KUKA KRL program: EPS_2_251674_SAN01_A_20251204014854.src

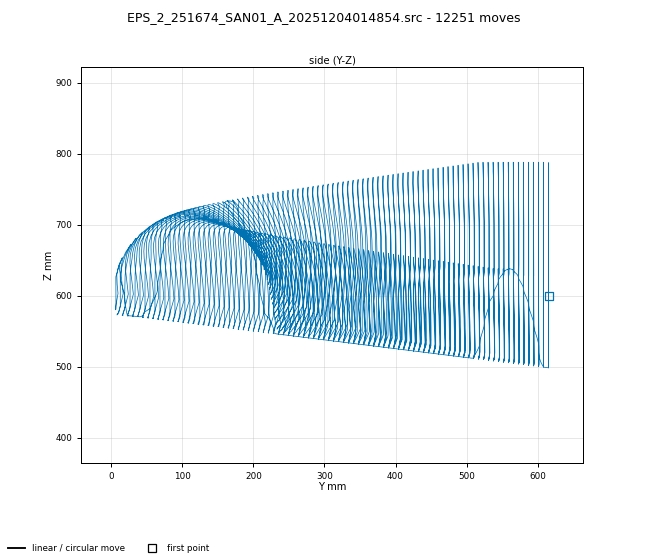
[picture p0: tool path of EPS_2_251674_SAN01_A_20251204014854.src, 12251 of 12253 moves have a stored position in this frame; points joined in program order, loops and branches not executed]
&ACCESS RVP
&REL 4
&COMMENT QRS 19112012
&PARAM EDITMASK = *
DEF PART()
EXT BAS (BAS_COMMAND :IN,REAL :IN )
INT I
BAS (#INITMOV,0 )

;KUKA QRS Post kuka4.cps  Date:22-06-2017 !

File_ID=2937

QRS_PRE_INIT()

;Init var - Until changes are made in qrs_pre_init
Outlet_Square_prg=0
Inlet_1_Square_prg=0
Inlet_2_Square_prg=0
Inlet_3_Square_prg=0
Inlet_4_Square_prg=0
Inlet_5_Square_prg=0

Outlet_1={X 0.000, Y 519.550, Z 713.000, B 0.000, E1 0.000 }
Inlet_1={X 0.000, Y 537.700, Z 427.500, B 0.000, E1 111.000 }
Outlet_1_type=150
Inlet_1_type=201
;QRS#1=Sidecore dimensions
;QRS#2=150-6" PVC SDR 28
;QRS#3=200-8" PVC SDR 35
;QRS#4=
;QRS#5=
;QRS#6=
;QRS#7=
;QRS#8=
;QRS#9=10-06 PSX
;QRS#10=12-08 PSX
;QRS#11=
;QRS#12=
;QRS#13=
;QRS#14=
;QRS#15=
;QRS#16=1220x127x1067 3,5'
;QRS#17=EPS Height
;QRS#18=788
;QRS#19=*
;QRS#20= UPDATED VERSION 22-06-2017
;QRS#21=*
Outlet_Square=070
Inlet_1_Square=0100
Inlet_2_Square=0
Inlet_3_Square=0
Inlet_4_Square=0
Inlet_5_Square=0
Mill_Square=1
Outlet_Square_Prg=203
Inlet_1_Square_prg=204

QRS_INIT()

$ADVANCE=5

; T1
PTP {E1 173.59,E2 173.59}
PTP {X 0,Y 615.512,A -85,B 0,C 180,E1 173.59,E2 173.59,E3 0,E4 0,E5 0,E6 0}
QRS_SPEED_INIT()
LIN {X 0,Y 615.512,Z 600,A -85,B 0,C 180,E1 173.59,E2 173.59,E3 0,E4 0,E5 0,E6 0} C_VEL
LIN {X 0,Y 615.512,Z 508.679,A -85,B 0,C 180,E1 173.59,E2 173.59} C_VEL
LIN {X 0,Y 615.512,Z 500.505,A -85,B 0,C 180,E1 173.59,E2 173.59} C_VEL
LIN {X 0,Y 615.495,Z 498.505,A -85,B 0,C 180,E1 173.404,E2 173.404} C_VEL
LIN {X 0,Y 615.498,Z 498.684,A -85,B 0,C 180,E1 171.091,E2 171.091} C_VEL
LIN {X 0,Y 615.497,Z 499.843,A -85,B 0,C 180,E1 170.967,E2 170.967} C_VEL
LIN {X 0,Y 615.499,Z 535.633,A -85,B 0,C 180,E1 170.511,E2 170.511} C_VEL
LIN {X 0,Y 615.498,Z 548.242,A -85,B 0,C 180,E1 170.221,E2 170.221} C_VEL
LIN {X 0,Y 615.498,Z 560.585,A -85,B 0,C 180,E1 169.806,E2 169.806} C_VEL
LIN {X 0,Y 615.498,Z 572.014,A -85,B 0,C 180,E1 169.287,E2 169.287} C_VEL
LIN {X 0,Y 615.494,Z 583.164,A -85,B 0,C 180,E1 168.64,E2 168.64} C_VEL
LIN {X 0,Y 615.498,Z 593.556,A -85,B 0,C 180,E1 167.888,E2 167.888} C_VEL
LIN {X 0,Y 615.498,Z 602.092,A -85,B 0,C 180,E1 167.134,E2 167.134} C_VEL
LIN {X 0,Y 615.498,Z 611.332,A -85,B 0,C 180,E1 166.126,E2 166.126} C_VEL
LIN {X 0,Y 615.498,Z 618.787,A -85,B 0,C 180,E1 165.113,E2 165.113} C_VEL
LIN {X 0,Y 615.496,Z 624.756,A -85,B 0,C 180,E1 164.095,E2 164.095} C_VEL
LIN {X 0,Y 615.496,Z 629.436,A -85,B 0,C 180,E1 163.072,E2 163.072} C_VEL
LIN {X 0,Y 615.495,Z 632.975,A -85,B 0,C 180,E1 162.043,E2 162.043} C_VEL
LIN {X 0,Y 615.497,Z 634.719,A -85,B 0,C 180,E1 161.354,E2 161.354} C_VEL
LIN {X 0,Y 615.495,Z 636.035,A -85,B 0,C 180,E1 160.662,E2 160.662} C_VEL
LIN {X 0,Y 615.493,Z 637.28,A -85,B 0,C 180,E1 159.438,E2 159.438} C_VEL
LIN {X 0,Y 615.499,Z 637.302,A -85,B 0,C 180,E1 158.568,E2 158.568} C_VEL
LIN {X 0,Y 615.491,Z 636.585,A -85,B 0,C 180,E1 157.65,E2 157.65} C_VEL
LIN {X 0,Y 615.494,Z 634.477,A -85,B 0,C 180,E1 156.444,E2 156.444} C_VEL
LIN {X 0,Y 615.496,Z 631.396,A -85,B 0,C 180,E1 155.369,E2 155.369} C_VEL
LIN {X 0,Y 615.494,Z 627.053,A -85,B 0,C 180,E1 154.284,E2 154.284} C_VEL
LIN {X 0,Y 615.498,Z 621.628,A -85,B 0,C 180,E1 153.254,E2 153.254} C_VEL
LIN {X 0,Y 615.494,Z 615.11,A -85,B 0,C 180,E1 152.27,E2 152.27} C_VEL
LIN {X 0,Y 615.497,Z 607.528,A -85,B 0,C 180,E1 151.342,E2 151.342} C_VEL
LIN {X 0,Y 615.498,Z 599.104,A -85,B 0,C 180,E1 150.496,E2 150.496} C_VEL
LIN {X 0,Y 615.495,Z 588.703,A -85,B 0,C 180,E1 149.651,E2 149.651} C_VEL
LIN {X 0,Y 615.497,Z 577.291,A -85,B 0,C 180,E1 148.91,E2 148.91} C_VEL
LIN {X 0,Y 615.498,Z 565.584,A -85,B 0,C 180,E1 148.315,E2 148.315} C_VEL
LIN {X 0,Y 615.496,Z 552.815,A -85,B 0,C 180,E1 147.828,E2 147.828} C_VEL
LIN {X 0,Y 615.497,Z 539.404,A -85,B 0,C 180,E1 147.47,E2 147.47} C_VEL
LIN {X 0,Y 615.497,Z 525.299,A -85,B 0,C 180,E1 147.251,E2 147.251} C_VEL
LIN {X 0,Y 615.496,Z 499.662,A -85,B 0,C 180,E1 146.935,E2 146.935} C_VEL
LIN {X 0,Y 615.495,Z 498.663,A -85,B 0,C 180,E1 146.813,E2 146.813} C_VEL
LIN {X 0,Y 615.487,Z 498.499,A -85,B 0,C 180,E1 144.164,E2 144.164} C_VEL
LIN {X 0,Y 615.478,Z 498.497,A -85,B 0,C 180,E1 141.93,E2 141.93} C_VEL
LIN {X 0,Y 615.482,Z 498.497,A -85,B 0,C 180,E1 139.393,E2 139.393} C_VEL
LIN {X 0,Y 615.485,Z 498.512,A -85,B 0,C 180,E1 136.755,E2 136.755} C_VEL
LIN {X 0,Y 615.482,Z 498.498,A -85,B 0,C 180,E1 133.996,E2 133.996} C_VEL
LIN {X 0,Y 615.483,Z 498.495,A -85,B 0,C 180,E1 131.473,E2 131.473} C_VEL
LIN {X 0,Y 615.482,Z 498.505,A -85,B 0,C 180,E1 128.904,E2 128.904} C_VEL
LIN {X 0,Y 615.491,Z 498.509,A -85,B 0,C 180,E1 126.423,E2 126.423} C_VEL
LIN {X 0,Y 615.479,Z 498.496,A -85,B 0,C 180,E1 123.532,E2 123.532} C_VEL
LIN {X 0,Y 615.48,Z 498.503,A -85,B 0,C 180,E1 120.919,E2 120.919} C_VEL
LIN {X 0,Y 615.496,Z 498.512,A -85,B 0,C 180,E1 118.451,E2 118.451} C_VEL
LIN {X 0,Y 615.477,Z 498.496,A -85,B 0,C 180,E1 115.566,E2 115.566} C_VEL
LIN {X 0,Y 615.482,Z 498.503,A -85,B 0,C 180,E1 112.844,E2 112.844} C_VEL
LIN {X 0,Y 615.489,Z 498.502,A -85,B 0,C 180,E1 110.032,E2 110.032} C_VEL
LIN {X 0,Y 615.485,Z 498.495,A -85,B 0,C 180,E1 107.27,E2 107.27} C_VEL
LIN {X 0,Y 615.484,Z 498.51,A -85,B 0,C 180,E1 104.549,E2 104.549} C_VEL
LIN {X 0,Y 615.485,Z 498.5,A -85,B 0,C 180,E1 101.861,E2 101.861} C_VEL
LIN {X 0,Y 615.486,Z 498.495,A -85,B 0,C 180,E1 99.199,E2 99.199} C_VEL
LIN {X 0,Y 615.477,Z 498.509,A -85,B 0,C 180,E1 96.557,E2 96.557} C_VEL
LIN {X 0,Y 615.487,Z 498.503,A -85,B 0,C 180,E1 93.928,E2 93.928} C_VEL
LIN {X 0,Y 615.48,Z 498.496,A -85,B 0,C 180,E1 91.309,E2 91.309} C_VEL
LIN {X 0,Y 615.483,Z 498.502,A -85,B 0,C 180,E1 88.691,E2 88.691} C_VEL
LIN {X 0,Y 615.496,Z 498.507,A -85,B 0,C 180,E1 86.072,E2 86.072} C_VEL
LIN {X 0,Y 615.477,Z 498.497,A -85,B 0,C 180,E1 83.435,E2 83.435} C_VEL
LIN {X 0,Y 615.486,Z 498.497,A -85,B 0,C 180,E1 80.801,E2 80.801} C_VEL
LIN {X 0,Y 615.489,Z 498.514,A -85,B 0,C 180,E1 78.139,E2 78.139} C_VEL
LIN {X 0,Y 615.476,Z 498.499,A -85,B 0,C 180,E1 75.451,E2 75.451} C_VEL
LIN {X 0,Y 615.485,Z 498.498,A -85,B 0,C 180,E1 72.73,E2 72.73} C_VEL
LIN {X 0,Y 615.495,Z 498.509,A -85,B 0,C 180,E1 69.968,E2 69.968} C_VEL
LIN {X 0,Y 615.48,Z 498.496,A -85,B 0,C 180,E1 67.156,E2 67.156} C_VEL
LIN {X 0,Y 615.479,Z 498.504,A -85,B 0,C 180,E1 64.434,E2 64.434} C_VEL
LIN {X 0,Y 615.487,Z 498.513,A -85,B 0,C 180,E1 62.086,E2 62.086} C_VEL
LIN {X 0,Y 615.499,Z 498.506,A -85,B 0,C 180,E1 59.841,E2 59.841} C_VEL
LIN {X 0,Y 615.481,Z 498.502,A -85,B 0,C 180,E1 57.543,E2 57.543} C_VEL
LIN {X 0,Y 615.478,Z 498.497,A -85,B 0,C 180,E1 55.185,E2 55.185} C_VEL
LIN {X 0,Y 615.491,Z 498.494,A -85,B 0,C 180,E1 52.759,E2 52.759} C_VEL
LIN {X 0,Y 615.497,Z 498.513,A -85,B 0,C 180,E1 49.911,E2 49.911} C_VEL
LIN {X 0,Y 615.485,Z 498.494,A -85,B 0,C 180,E1 46.953,E2 46.953} C_VEL
LIN {X 0,Y 615.478,Z 498.508,A -85,B 0,C 180,E1 44.151,E2 44.151} C_VEL
LIN {X 0,Y 615.482,Z 498.503,A -85,B 0,C 180,E1 41.475,E2 41.475} C_VEL
LIN {X 0,Y 615.484,Z 498.495,A -85,B 0,C 180,E1 38.905,E2 38.905} C_VEL
LIN {X 0,Y 615.481,Z 498.499,A -85,B 0,C 180,E1 36.426,E2 36.426} C_VEL
LIN {X 0,Y 615.486,Z 498.506,A -85,B 0,C 180,E1 33.536,E2 33.536} C_VEL
LIN {X 0,Y 615.483,Z 498.495,A -85,B 0,C 180,E1 30.92,E2 30.92} C_VEL
LIN {X 0,Y 615.483,Z 498.497,A -85,B 0,C 180,E1 28.452,E2 28.452} C_VEL
LIN {X 0,Y 615.493,Z 498.508,A -85,B 0,C 180,E1 25.573,E2 25.573} C_VEL
LIN {X 0,Y 615.482,Z 498.496,A -85,B 0,C 180,E1 22.845,E2 22.845} C_VEL
LIN {X 0,Y 615.477,Z 498.505,A -85,B 0,C 180,E1 20.033,E2 20.033} C_VEL
LIN {X 0,Y 615.479,Z 498.504,A -85,B 0,C 180,E1 17.271,E2 17.271} C_VEL
LIN {X 0,Y 615.488,Z 498.494,A -85,B 0,C 180,E1 14.549,E2 14.549} C_VEL
LIN {X 0,Y 615.479,Z 498.508,A -85,B 0,C 180,E1 11.861,E2 11.861} C_VEL
LIN {X 0,Y 615.479,Z 498.504,A -85,B 0,C 180,E1 9.199,E2 9.199} C_VEL
LIN {X 0,Y 615.491,Z 498.493,A -85,B 0,C 180,E1 6.557,E2 6.557} C_VEL
LIN {X 0,Y 615.475,Z 498.505,A -85,B 0,C 180,E1 3.929,E2 3.929} C_VEL
LIN {X 0,Y 615.484,Z 498.508,A -85,B 0,C 180,E1 1.309,E2 1.309} C_VEL
LIN {X 0,Y 615.485,Z 498.495,A -85,B 0,C 180,E1 -1.308,E2 -1.308} C_VEL
LIN {X 0,Y 615.477,Z 498.5,A -85,B 0,C 180,E1 -3.928,E2 -3.928} C_VEL
LIN {X 0,Y 615.49,Z 498.513,A -85,B 0,C 180,E1 -6.591,E2 -6.591} C_VEL
LIN {X 0,Y 615.479,Z 498.499,A -85,B 0,C 180,E1 -9.199,E2 -9.199} C_VEL
LIN {X 0,Y 615.479,Z 498.497,A -85,B 0,C 180,E1 -11.861,E2 -11.861} C_VEL
LIN {X 0,Y 615.488,Z 498.513,A -85,B 0,C 180,E1 -14.549,E2 -14.549} C_VEL
LIN {X 0,Y 615.478,Z 498.499,A -85,B 0,C 180,E1 -17.271,E2 -17.271} C_VEL
LIN {X 0,Y 615.477,Z 498.499,A -85,B 0,C 180,E1 -20.033,E2 -20.033} C_VEL
LIN {X 0,Y 615.482,Z 498.51,A -85,B 0,C 180,E1 -22.845,E2 -22.845} C_VEL
LIN {X 0,Y 615.493,Z 498.493,A -85,B 0,C 180,E1 -25.715,E2 -25.715} C_VEL
LIN {X 0,Y 615.487,Z 498.513,A -85,B 0,C 180,E1 -28.658,E2 -28.658} C_VEL
LIN {X 0,Y 615.478,Z 498.505,A -85,B 0,C 180,E1 -31.087,E2 -31.087} C_VEL
LIN {X 0,Y 615.485,Z 498.496,A -85,B 0,C 180,E1 -33.536,E2 -33.536} C_VEL
LIN {X 0,Y 615.486,Z 498.494,A -85,B 0,C 180,E1 -35.835,E2 -35.835} C_VEL
LIN {X 0,Y 615.478,Z 498.498,A -85,B 0,C 180,E1 -38.069,E2 -38.069} C_VEL
LIN {X 0,Y 615.482,Z 498.508,A -85,B 0,C 180,E1 -40.607,E2 -40.607} C_VEL
LIN {X 0,Y 615.477,Z 498.504,A -85,B 0,C 180,E1 -43.245,E2 -43.245} C_VEL
LIN {X 0,Y 615.482,Z 498.495,A -85,B 0,C 180,E1 -46.003,E2 -46.003} C_VEL
LIN {X 0,Y 615.483,Z 498.504,A -85,B 0,C 180,E1 -48.527,E2 -48.527} C_VEL
LIN {X 0,Y 615.479,Z 498.51,A -85,B 0,C 180,E1 -51.096,E2 -51.096} C_VEL
LIN {X 0,Y 615.484,Z 498.497,A -85,B 0,C 180,E1 -53.576,E2 -53.576} C_VEL
LIN {X 0,Y 615.479,Z 498.502,A -85,B 0,C 180,E1 -56.467,E2 -56.467} C_VEL
LIN {X 0,Y 615.477,Z 498.514,A -85,B 0,C 180,E1 -59.08,E2 -59.08} C_VEL
LIN {X 0,Y 615.482,Z 498.5,A -85,B 0,C 180,E1 -61.551,E2 -61.551} C_VEL
LIN {X 0,Y 615.495,Z 498.704,A -85,B 0,C 180,E1 -63.104,E2 -63.104} C_VEL
LIN {X 0,Y 615.495,Z 501.655,A -85,B 0,C 180,E1 -63.557,E2 -63.557} C_VEL
LIN {X 0,Y 615.481,Z 521.157,A -85,B 0,C 180,E1 -66.217,E2 -66.217} C_VEL
LIN {X 0,Y 615.497,Z 541.369,A -85,B 0,C 180,E1 -68.92,E2 -68.92} C_VEL
LIN {X 0,Y 615.492,Z 563.931,A -85,B 0,C 180,E1 -71.882,E2 -71.882} C_VEL
LIN {X 0,Y 615.489,Z 586.305,A -85,B 0,C 180,E1 -74.774,E2 -74.774} C_VEL
LIN {X 0,Y 615.477,Z 608.735,A -85,B 0,C 180,E1 -77.637,E2 -77.637} C_VEL
LIN {X 0,Y 615.491,Z 626.165,A -85,B 0,C 180,E1 -79.827,E2 -79.827} C_VEL
LIN {X 0,Y 615.492,Z 628.081,A -85,B 0,C 180,E1 -79.889,E2 -79.889} C_VEL
LIN {X 0,Y 615.489,Z 704.946,A -85,B 0,C 180,E1 -80.801,E2 -80.801} C_VEL
LIN {X 0,Y 615.496,Z 714.698,A -85,B 0,C 180,E1 -81.009,E2 -81.009} C_VEL
LIN {X 0,Y 615.499,Z 725.155,A -85,B 0,C 180,E1 -81.34,E2 -81.34} C_VEL
LIN {X 0,Y 615.498,Z 735.429,A -85,B 0,C 180,E1 -81.794,E2 -81.794} C_VEL
LIN {X 0,Y 615.488,Z 745.201,A -85,B 0,C 180,E1 -82.372,E2 -82.372} C_VEL
LIN {X 0,Y 615.495,Z 752.935,A -85,B 0,C 180,E1 -82.942,E2 -82.942} C_VEL
LIN {X 0,Y 615.497,Z 760.335,A -85,B 0,C 180,E1 -83.608,E2 -83.608} C_VEL
LIN {X 0,Y 615.498,Z 767.738,A -85,B 0,C 180,E1 -84.43,E2 -84.43} C_VEL
LIN {X 0,Y 615.498,Z 773.533,A -85,B 0,C 180,E1 -85.251,E2 -85.251} C_VEL
LIN {X 0,Y 615.493,Z 778.101,A -85,B 0,C 180,E1 -86.072,E2 -86.072} C_VEL
LIN {X 0,Y 615.493,Z 781.068,A -85,B 0,C 180,E1 -86.727,E2 -86.727} C_VEL
LIN {X 0,Y 615.495,Z 783.356,A -85,B 0,C 180,E1 -87.382,E2 -87.382} C_VEL
LIN {X 0,Y 615.495,Z 785.086,A -85,B 0,C 180,E1 -88.037,E2 -88.037} C_VEL
LIN {X 0,Y 615.494,Z 786.33,A -85,B 0,C 180,E1 -88.691,E2 -88.691} C_VEL
LIN {X 0,Y 615.493,Z 787.104,A -85,B 0,C 180,E1 -89.346,E2 -89.346} C_VEL
LIN {X 0,Y 615.491,Z 787.389,A -85,B 0,C 180,E1 -90,E2 -90} C_VEL
LIN {X 0,Y 615.494,Z 787.104,A -85,B 0,C 180,E1 -90.654,E2 -90.654} C_VEL
LIN {X 0,Y 615.494,Z 786.33,A -85,B 0,C 180,E1 -91.308,E2 -91.308} C_VEL
LIN {X 0,Y 615.495,Z 785.086,A -85,B 0,C 180,E1 -91.963,E2 -91.963} C_VEL
LIN {X 0,Y 615.493,Z 782.22,A -85,B 0,C 180,E1 -92.945,E2 -92.945} C_VEL
LIN {X 0,Y 615.492,Z 779.604,A -85,B 0,C 180,E1 -93.601,E2 -93.601} C_VEL
LIN {X 0,Y 615.497,Z 774.483,A -85,B 0,C 180,E1 -94.584,E2 -94.584} C_VEL
LIN {X 0,Y 615.495,Z 768.969,A -85,B 0,C 180,E1 -95.405,E2 -95.405} C_VEL
LIN {X 0,Y 615.498,Z 762.02,A -85,B 0,C 180,E1 -96.227,E2 -96.227} C_VEL
LIN {X 0,Y 615.496,Z 754.86,A -85,B 0,C 180,E1 -96.901,E2 -96.901} C_VEL
LIN {X 0,Y 615.485,Z 747.626,A -85,B 0,C 180,E1 -97.463,E2 -97.463} C_VEL
LIN {X 0,Y 615.497,Z 739.872,A -85,B 0,C 180,E1 -97.958,E2 -97.958} C_VEL
LIN {X 0,Y 615.499,Z 731.918,A -85,B 0,C 180,E1 -98.371,E2 -98.371} C_VEL
LIN {X 0,Y 615.497,Z 722.761,A -85,B 0,C 180,E1 -98.743,E2 -98.743} C_VEL
LIN {X 0,Y 615.496,Z 714.702,A -85,B 0,C 180,E1 -98.991,E2 -98.991} C_VEL
LIN {X 0,Y 615.489,Z 704.952,A -85,B 0,C 180,E1 -99.198,E2 -99.198} C_VEL
LIN {X 0,Y 615.492,Z 626.948,A -85,B 0,C 180,E1 -100.132,E2 -100.132} C_VEL
LIN {X 0,Y 615.489,Z 625.928,A -85,B 0,C 180,E1 -100.194,E2 -100.194} C_VEL
LIN {X 0,Y 615.488,Z 603.458,A -85,B 0,C 180,E1 -103.033,E2 -103.033} C_VEL
LIN {X 0,Y 615.486,Z 581.024,A -85,B 0,C 180,E1 -105.905,E2 -105.905} C_VEL
LIN {X 0,Y 615.481,Z 559.887,A -85,B 0,C 180,E1 -108.646,E2 -108.646} C_VEL
LIN {X 0,Y 615.492,Z 538.723,A -85,B 0,C 180,E1 -111.431,E2 -111.431} C_VEL
LIN {X 0,Y 615.494,Z 517.542,A -85,B 0,C 180,E1 -114.271,E2 -114.271} C_VEL
LIN {X 0,Y 615.495,Z 498.824,A -85,B 0,C 180,E1 -116.858,E2 -116.858} C_VEL
LIN {X 0,Y 615.491,Z 498.508,A -85,B 0,C 180,E1 -117.176,E2 -117.176} C_VEL
LIN {X 0,Y 615.499,Z 498.492,A -85,B 0,C 180,E1 -120.159,E2 -120.159} C_VEL
LIN {X 0,Y 615.481,Z 498.501,A -85,B 0,C 180,E1 -122.457,E2 -122.457} C_VEL
LIN {X 0,Y 615.479,Z 498.511,A -85,B 0,C 180,E1 -124.815,E2 -124.815} C_VEL
LIN {X 0,Y 615.492,Z 498.505,A -85,B 0,C 180,E1 -127.241,E2 -127.241} C_VEL
LIN {X 0,Y 615.489,Z 498.494,A -85,B 0,C 180,E1 -130.089,E2 -130.089} C_VEL
LIN {X 0,Y 615.497,Z 498.51,A -85,B 0,C 180,E1 -133.048,E2 -133.048} C_VEL
LIN {X 0,Y 615.482,Z 498.496,A -85,B 0,C 180,E1 -136.002,E2 -136.002} C_VEL
LIN {X 0,Y 615.491,Z 498.513,A -85,B 0,C 180,E1 -138.904,E2 -138.904} C_VEL
LIN {X 0,Y 615.496,Z 498.507,A -85,B 0,C 180,E1 -141.096,E2 -141.096} C_VEL
LIN {X 0,Y 615.481,Z 498.498,A -85,B 0,C 180,E1 -143.575,E2 -143.575} C_VEL
LIN {X 0,Y 615.479,Z 498.496,A -85,B 0,C 180,E1 -145.978,E2 -145.978} C_VEL
LIN {X 0,Y 615.485,Z 498.498,A -85,B 0,C 180,E1 -148.315,E2 -148.315} C_VEL
LIN {X 0,Y 615.482,Z 498.505,A -85,B 0,C 180,E1 -150.594,E2 -150.594} C_VEL
LIN {X 0,Y 615.498,Z 498.511,A -85,B 0,C 180,E1 -152.95,E2 -152.95} C_VEL
LIN {X 0,Y 615.478,Z 498.497,A -85,B 0,C 180,E1 -155.728,E2 -155.728} C_VEL
LIN {X 0,Y 615.477,Z 498.497,A -85,B 0,C 180,E1 -157.863,E2 -157.863} C_VEL
LIN {X 0,Y 615.486,Z 498.507,A -85,B 0,C 180,E1 -160.662,E2 -160.662} C_VEL
LIN {X 0,Y 615.485,Z 498.497,A -85,B 0,C 180,E1 -163.565,E2 -163.565} C_VEL
LIN {X 0,Y 615.476,Z 498.498,A -85,B 0,C 180,E1 -166.126,E2 -166.126} C_VEL
LIN {X 0,Y 615.49,Z 498.512,A -85,B 0,C 180,E1 -168.807,E2 -168.807} C_VEL
LIN {X 0,Y 615.491,Z 498.497,A -85,B 0,C 180,E1 -171.464,E2 -171.464} C_VEL
LIN {X 0,Y 615.478,Z 498.498,A -85,B 0,C 180,E1 -174.102,E2 -174.102} C_VEL
LIN {X 0,Y 615.496,Z 498.509,A -85,B 0,C 180,E1 -176.727,E2 -176.727} C_VEL
LIN {X 0,Y 615.488,Z 498.5,A -85,B 0,C 180,E1 -179.346,E2 -179.346} C_VEL
LIN {X 0,Y 615.477,Z 498.497,A -85,B 0,C 180,E1 -181.963,E2 -181.963} C_VEL
LIN {X 0,Y 615.495,Z 498.505,A -85,B 0,C 180,E1 -184.585,E2 -184.585} C_VEL
LIN {X 0,Y 615.495,Z 498.505,A -85,B 0,C 180,E1 -186.596,E2 -186.596} C_VEL
LIN {X 0,Y 614.805,Z 498.657,A -85,B 0,C 180,E1 -186.961,E2 -186.961} C_VEL
LIN {X 0,Y 609.123,Z 499.426,A -85,B 0,C 180,E1 -188.104,E2 -188.104} C_VEL
LIN {X 0,Y 608.459,Z 499.504,A -85,B 0,C 180,E1 -188.474,E2 -188.474} C_VEL
LIN {X 0,Y 608.519,Z 499.771,A -85,B 0,C 180,E1 -188.824,E2 -188.824} C_VEL
LIN {X 0,Y 608.563,Z 500.764,A -85,B 0,C 180,E1 -188.907,E2 -188.907} C_VEL
LIN {X 0,Y 608.557,Z 535.292,A -85,B 0,C 180,E1 -189.347,E2 -189.347} C_VEL
LIN {X 0,Y 608.553,Z 548.8,A -85,B 0,C 180,E1 -189.661,E2 -189.661} C_VEL
LIN {X 0,Y 608.52,Z 561.542,A -85,B 0,C 180,E1 -190.103,E2 -190.103} C_VEL
LIN {X 0,Y 608.501,Z 573.22,A -85,B 0,C 180,E1 -190.649,E2 -190.649} C_VEL
LIN {X 0,Y 608.484,Z 584.526,A -85,B 0,C 180,E1 -191.324,E2 -191.324} C_VEL
LIN {X 0,Y 608.48,Z 594.764,A -85,B 0,C 180,E1 -192.084,E2 -192.084} C_VEL
LIN {X 0,Y 608.465,Z 604.82,A -85,B 0,C 180,E1 -193.017,E2 -193.017} C_VEL
LIN {X 0,Y 608.461,Z 613.689,A -85,B 0,C 180,E1 -194.038,E2 -194.038} C_VEL
LIN {X 0,Y 608.442,Z 620.782,A -85,B 0,C 180,E1 -195.064,E2 -195.064} C_VEL
LIN {X 0,Y 608.458,Z 626.458,A -85,B 0,C 180,E1 -196.094,E2 -196.094} C_VEL
LIN {X 0,Y 608.455,Z 630.897,A -85,B 0,C 180,E1 -197.13,E2 -197.13} C_VEL
LIN {X 0,Y 608.422,Z 634.214,A -85,B 0,C 180,E1 -198.173,E2 -198.173} C_VEL
LIN {X 0,Y 608.436,Z 635.847,A -85,B 0,C 180,E1 -198.871,E2 -198.871} C_VEL
LIN {X 0,Y 608.417,Z 637.008,A -85,B 0,C 180,E1 -199.572,E2 -199.572} C_VEL
LIN {X 0,Y 608.435,Z 637.919,A -85,B 0,C 180,E1 -200.674,E2 -200.674} C_VEL
LIN {X 0,Y 608.418,Z 637.793,A -85,B 0,C 180,E1 -201.694,E2 -201.694} C_VEL
LIN {X 0,Y 608.418,Z 637.064,A -85,B 0,C 180,E1 -202.47,E2 -202.47} C_VEL
LIN {X 0,Y 608.421,Z 636.041,A -85,B 0,C 180,E1 -203.125,E2 -203.125} C_VEL
LIN {X 0,Y 608.427,Z 633.605,A -85,B 0,C 180,E1 -204.145,E2 -204.145} C_VEL
LIN {X 0,Y 608.442,Z 629.579,A -85,B 0,C 180,E1 -205.302,E2 -205.302} C_VEL
LIN {X 0,Y 608.452,Z 624.363,A -85,B 0,C 180,E1 -206.404,E2 -206.404} C_VEL
LIN {X 0,Y 608.443,Z 617.567,A -85,B 0,C 180,E1 -207.519,E2 -207.519} C_VEL
LIN {X 0,Y 608.465,Z 610.528,A -85,B 0,C 180,E1 -208.443,E2 -208.443} C_VEL
LIN {X 0,Y 608.462,Z 601.547,A -85,B 0,C 180,E1 -209.4,E2 -209.4} C_VEL
LIN {X 0,Y 608.487,Z 590.988,A -85,B 0,C 180,E1 -210.305,E2 -210.305} C_VEL
LIN {X 0,Y 608.493,Z 580.516,A -85,B 0,C 180,E1 -211.025,E2 -211.025} C_VEL
LIN {X 0,Y 608.507,Z 569.004,A -85,B 0,C 180,E1 -211.654,E2 -211.654} C_VEL
LIN {X 0,Y 608.52,Z 556.674,A -85,B 0,C 180,E1 -212.174,E2 -212.174} C_VEL
LIN {X 0,Y 608.549,Z 543.589,A -85,B 0,C 180,E1 -212.569,E2 -212.569} C_VEL
LIN {X 0,Y 608.548,Z 530.272,A -85,B 0,C 180,E1 -212.822,E2 -212.822} C_VEL
LIN {X 0,Y 608.583,Z 500.534,A -85,B 0,C 180,E1 -213.193,E2 -213.193} C_VEL
LIN {X 0,Y 608.485,Z 499.565,A -85,B 0,C 180,E1 -213.323,E2 -213.323} C_VEL
LIN {X 0,Y 608.472,Z 499.498,A -85,B 0,C 180,E1 -216.091,E2 -216.091} C_VEL
LIN {X 0,Y 608.465,Z 499.499,A -85,B 0,C 180,E1 -218.589,E2 -218.589} C_VEL
LIN {X 0,Y 608.467,Z 499.509,A -85,B 0,C 180,E1 -221.344,E2 -221.344} C_VEL
LIN {X 0,Y 608.448,Z 499.5,A -85,B 0,C 180,E1 -224.264,E2 -224.264} C_VEL
LIN {X 0,Y 608.454,Z 499.504,A -85,B 0,C 180,E1 -227.042,E2 -227.042} C_VEL
LIN {X 0,Y 608.456,Z 499.505,A -85,B 0,C 180,E1 -229.698,E2 -229.698} C_VEL
LIN {X 0,Y 608.47,Z 499.497,A -85,B 0,C 180,E1 -232.255,E2 -232.255} C_VEL
LIN {X 0,Y 608.443,Z 499.505,A -85,B 0,C 180,E1 -235.096,E2 -235.096} C_VEL
LIN {X 0,Y 608.471,Z 499.501,A -85,B 0,C 180,E1 -237.907,E2 -237.907} C_VEL
LIN {X 0,Y 608.463,Z 499.499,A -85,B 0,C 180,E1 -240.221,E2 -240.221} C_VEL
LIN {X 0,Y 608.481,Z 499.497,A -85,B 0,C 180,E1 -242.793,E2 -242.793} C_VEL
LIN {X 0,Y 608.485,Z 499.501,A -85,B 0,C 180,E1 -245.847,E2 -245.847} C_VEL
LIN {X 0,Y 608.469,Z 499.498,A -85,B 0,C 180,E1 -248.309,E2 -248.309} C_VEL
LIN {X 0,Y 608.455,Z 499.502,A -85,B 0,C 180,E1 -251.131,E2 -251.131} C_VEL
LIN {X 0,Y 608.463,Z 499.504,A -85,B 0,C 180,E1 -253.907,E2 -253.907} C_VEL
LIN {X 0,Y 608.465,Z 499.498,A -85,B 0,C 180,E1 -256.644,E2 -256.644} C_VEL
LIN {X 0,Y 608.461,Z 499.504,A -85,B 0,C 180,E1 -259.35,E2 -259.35} C_VEL
LIN {X 0,Y 608.479,Z 499.501,A -85,B 0,C 180,E1 -262.033,E2 -262.033} C_VEL
LIN {X 0,Y 608.46,Z 499.498,A -85,B 0,C 180,E1 -264.698,E2 -264.698} C_VEL
LIN {X 0,Y 608.47,Z 499.502,A -85,B 0,C 180,E1 -267.352,E2 -267.352} C_VEL
LIN {X 0,Y 608.482,Z 499.502,A -85,B 0,C 180,E1 -270,E2 -270} C_VEL
LIN {X 0,Y 608.469,Z 499.497,A -85,B 0,C 180,E1 -272.648,E2 -272.648} C_VEL
LIN {X 0,Y 608.461,Z 499.501,A -85,B 0,C 180,E1 -275.302,E2 -275.302} C_VEL
LIN {X 0,Y 608.481,Z 499.504,A -85,B 0,C 180,E1 -277.967,E2 -277.967} C_VEL
LIN {X 0,Y 608.459,Z 499.499,A -85,B 0,C 180,E1 -280.65,E2 -280.65} C_VEL
LIN {X 0,Y 608.468,Z 499.5,A -85,B 0,C 180,E1 -283.356,E2 -283.356} C_VEL
LIN {X 0,Y 608.461,Z 499.505,A -85,B 0,C 180,E1 -286.093,E2 -286.093} C_VEL
LIN {X 0,Y 608.454,Z 499.499,A -85,B 0,C 180,E1 -288.869,E2 -288.869} C_VEL
LIN {X 0,Y 608.469,Z 499.504,A -85,B 0,C 180,E1 -291.691,E2 -291.691} C_VEL
LIN {X 0,Y 608.456,Z 499.501,A -85,B 0,C 180,E1 -294.57,E2 -294.57} C_VEL
LIN {X 0,Y 608.481,Z 499.496,A -85,B 0,C 180,E1 -297.207,E2 -297.207} C_VEL
LIN {X 0,Y 608.468,Z 499.509,A -85,B 0,C 180,E1 -299.971,E2 -299.971} C_VEL
LIN {X 0,Y 608.455,Z 499.499,A -85,B 0,C 180,E1 -302.879,E2 -302.879} C_VEL
LIN {X 0,Y 608.435,Z 499.502,A -85,B 0,C 180,E1 -305.277,E2 -305.277} C_VEL
LIN {X 0,Y 608.473,Z 499.502,A -85,B 0,C 180,E1 -307.745,E2 -307.745} C_VEL
LIN {X 0,Y 608.453,Z 499.506,A -85,B 0,C 180,E1 -310.329,E2 -310.329} C_VEL
LIN {X 0,Y 608.453,Z 499.499,A -85,B 0,C 180,E1 -312.959,E2 -312.959} C_VEL
LIN {X 0,Y 608.449,Z 499.504,A -85,B 0,C 180,E1 -315.736,E2 -315.736} C_VEL
LIN {X 0,Y 608.457,Z 499.502,A -85,B 0,C 180,E1 -318.657,E2 -318.657} C_VEL
LIN {X 0,Y 608.466,Z 499.498,A -85,B 0,C 180,E1 -321.411,E2 -321.411} C_VEL
LIN {X 0,Y 608.473,Z 499.503,A -85,B 0,C 180,E1 -323.949,E2 -323.949} C_VEL
LIN {X 0,Y 608.462,Z 499.507,A -85,B 0,C 180,E1 -326.329,E2 -326.329} C_VEL
LIN {X 0,Y 608.471,Z 499.5,A -85,B 0,C 180,E1 -328.727,E2 -328.727} C_VEL
LIN {X 0,Y 608.471,Z 499.497,A -85,B 0,C 180,E1 -331.378,E2 -331.378} C_VEL
LIN {X 0,Y 608.479,Z 499.508,A -85,B 0,C 180,E1 -334.275,E2 -334.275} C_VEL
LIN {X 0,Y 608.448,Z 499.502,A -85,B 0,C 180,E1 -336.876,E2 -336.876} C_VEL
LIN {X 0,Y 608.458,Z 499.501,A -85,B 0,C 180,E1 -339.725,E2 -339.725} C_VEL
LIN {X 0,Y 608.445,Z 499.508,A -85,B 0,C 180,E1 -342.523,E2 -342.523} C_VEL
LIN {X 0,Y 608.473,Z 499.497,A -85,B 0,C 180,E1 -345.279,E2 -345.279} C_VEL
LIN {X 0,Y 608.456,Z 499.503,A -85,B 0,C 180,E1 -348,E2 -348} C_VEL
LIN {X 0,Y 608.462,Z 499.504,A -85,B 0,C 180,E1 -350.694,E2 -350.694} C_VEL
LIN {X 0,Y 608.467,Z 499.498,A -85,B 0,C 180,E1 -353.367,E2 -353.367} C_VEL
LIN {X 0,Y 608.445,Z 499.504,A -85,B 0,C 180,E1 -356.026,E2 -356.026} C_VEL
LIN {X 0,Y 608.467,Z 499.505,A -85,B 0,C 180,E1 -358.676,E2 -358.676} C_VEL
LIN {X 0,Y 608.468,Z 499.498,A -85,B 0,C 180,E1 -361.323,E2 -361.323} C_VEL
LIN {X 0,Y 608.448,Z 499.502,A -85,B 0,C 180,E1 -363.974,E2 -363.974} C_VEL
LIN {X 0,Y 608.466,Z 499.507,A -85,B 0,C 180,E1 -366.632,E2 -366.632} C_VEL
LIN {X 0,Y 608.462,Z 499.499,A -85,B 0,C 180,E1 -369.306,E2 -369.306} C_VEL
LIN {X 0,Y 608.457,Z 499.501,A -85,B 0,C 180,E1 -372,E2 -372} C_VEL
LIN {X 0,Y 608.472,Z 499.506,A -85,B 0,C 180,E1 -374.72,E2 -374.72} C_VEL
LIN {X 0,Y 608.445,Z 499.5,A -85,B 0,C 180,E1 -377.477,E2 -377.477} C_VEL
LIN {X 0,Y 608.458,Z 499.503,A -85,B 0,C 180,E1 -380.274,E2 -380.274} C_VEL
LIN {X 0,Y 608.449,Z 499.507,A -85,B 0,C 180,E1 -382.477,E2 -382.477} C_VEL
LIN {X 0,Y 608.451,Z 499.501,A -85,B 0,C 180,E1 -385.301,E2 -385.301} C_VEL
LIN {X 0,Y 608.443,Z 499.501,A -85,B 0,C 180,E1 -387.518,E2 -387.518} C_VEL
LIN {X 0,Y 608.464,Z 499.498,A -85,B 0,C 180,E1 -389.973,E2 -389.973} C_VEL
LIN {X 0,Y 608.458,Z 499.506,A -85,B 0,C 180,E1 -392.524,E2 -392.524} C_VEL
LIN {X 0,Y 608.451,Z 499.502,A -85,B 0,C 180,E1 -395.277,E2 -395.277} C_VEL
LIN {X 0,Y 608.463,Z 499.498,A -85,B 0,C 180,E1 -397.747,E2 -397.747} C_VEL
LIN {X 0,Y 608.446,Z 499.503,A -85,B 0,C 180,E1 -400.33,E2 -400.33} C_VEL
LIN {X 0,Y 608.448,Z 499.509,A -85,B 0,C 180,E1 -402.96,E2 -402.96} C_VEL
LIN {X 0,Y 608.459,Z 499.499,A -85,B 0,C 180,E1 -405.736,E2 -405.736} C_VEL
LIN {X 0,Y 608.459,Z 499.505,A -85,B 0,C 180,E1 -408.658,E2 -408.658} C_VEL
LIN {X 0,Y 608.465,Z 499.501,A -85,B 0,C 180,E1 -411.413,E2 -411.413} C_VEL
LIN {X 0,Y 608.472,Z 499.497,A -85,B 0,C 180,E1 -413.951,E2 -413.951} C_VEL
LIN {X 0,Y 608.459,Z 499.5,A -85,B 0,C 180,E1 -416.33,E2 -416.33} C_VEL
LIN {X 0,Y 608.475,Z 499.503,A -85,B 0,C 180,E1 -418.728,E2 -418.728} C_VEL
LIN {X 0,Y 608.468,Z 499.504,A -85,B 0,C 180,E1 -421.381,E2 -421.381} C_VEL
LIN {X 0,Y 608.498,Z 499.663,A -85,B 0,C 180,E1 -422.923,E2 -422.923} C_VEL
LIN {X 0,Y 608.659,Z 502.978,A -85,B 0,C 180,E1 -423.421,E2 -423.421} C_VEL
LIN {X 0,Y 608.606,Z 522.836,A -85,B 0,C 180,E1 -426.161,E2 -426.161} C_VEL
LIN {X 0,Y 608.571,Z 542.694,A -85,B 0,C 180,E1 -428.846,E2 -428.846} C_VEL
LIN {X 0,Y 608.544,Z 563.958,A -85,B 0,C 180,E1 -431.668,E2 -431.668} C_VEL
LIN {X 0,Y 608.487,Z 585.058,A -85,B 0,C 180,E1 -434.423,E2 -434.423} C_VEL
LIN {X 0,Y 608.488,Z 604.916,A -85,B 0,C 180,E1 -436.984,E2 -436.984} C_VEL
LIN {X 0,Y 608.472,Z 626.35,A -85,B 0,C 180,E1 -439.708,E2 -439.708} C_VEL
LIN {X 0,Y 608.525,Z 628.526,A -85,B 0,C 180,E1 -439.772,E2 -439.772} C_VEL
LIN {X 0,Y 608.499,Z 704.155,A -85,B 0,C 180,E1 -440.674,E2 -440.674} C_VEL
LIN {X 0,Y 608.519,Z 713.421,A -85,B 0,C 180,E1 -440.863,E2 -440.863} C_VEL
LIN {X 0,Y 608.49,Z 721.892,A -85,B 0,C 180,E1 -441.114,E2 -441.114} C_VEL
LIN {X 0,Y 608.501,Z 730.391,A -85,B 0,C 180,E1 -441.448,E2 -441.448} C_VEL
LIN {X 0,Y 608.497,Z 738.721,A -85,B 0,C 180,E1 -441.866,E2 -441.866} C_VEL
LIN {X 0,Y 608.467,Z 746.761,A -85,B 0,C 180,E1 -442.367,E2 -442.367} C_VEL
LIN {X 0,Y 608.454,Z 754.416,A -85,B 0,C 180,E1 -442.951,E2 -442.951} C_VEL
LIN {X 0,Y 608.452,Z 762.439,A -85,B 0,C 180,E1 -443.7,E2 -443.7} C_VEL
LIN {X 0,Y 608.46,Z 769.43,A -85,B 0,C 180,E1 -444.532,E2 -444.532} C_VEL
LIN {X 0,Y 608.447,Z 774.985,A -85,B 0,C 180,E1 -445.362,E2 -445.362} C_VEL
LIN {X 0,Y 608.446,Z 780.146,A -85,B 0,C 180,E1 -446.358,E2 -446.358} C_VEL
LIN {X 0,Y 608.448,Z 782.786,A -85,B 0,C 180,E1 -447.021,E2 -447.021} C_VEL
LIN {X 0,Y 608.44,Z 785.678,A -85,B 0,C 180,E1 -448.014,E2 -448.014} C_VEL
LIN {X 0,Y 608.446,Z 786.933,A -85,B 0,C 180,E1 -448.676,E2 -448.676} C_VEL
LIN {X 0,Y 608.436,Z 787.714,A -85,B 0,C 180,E1 -449.338,E2 -449.338} C_VEL
LIN {X 0,Y 608.431,Z 788,A -85,B 0,C 180,E1 -450,E2 -450} C_VEL
LIN {X 0,Y 608.436,Z 787.714,A -85,B 0,C 180,E1 -450.662,E2 -450.662} C_VEL
LIN {X 0,Y 608.446,Z 786.934,A -85,B 0,C 180,E1 -451.324,E2 -451.324} C_VEL
LIN {X 0,Y 608.44,Z 785.678,A -85,B 0,C 180,E1 -451.986,E2 -451.986} C_VEL
LIN {X 0,Y 608.448,Z 782.786,A -85,B 0,C 180,E1 -452.979,E2 -452.979} C_VEL
LIN {X 0,Y 608.446,Z 780.147,A -85,B 0,C 180,E1 -453.642,E2 -453.642} C_VEL
LIN {X 0,Y 608.447,Z 774.986,A -85,B 0,C 180,E1 -454.638,E2 -454.638} C_VEL
LIN {X 0,Y 608.46,Z 769.431,A -85,B 0,C 180,E1 -455.468,E2 -455.468} C_VEL
LIN {X 0,Y 608.455,Z 761.669,A -85,B 0,C 180,E1 -456.376,E2 -456.376} C_VEL
LIN {X 0,Y 608.454,Z 754.417,A -85,B 0,C 180,E1 -457.049,E2 -457.049} C_VEL
LIN {X 0,Y 608.467,Z 746.763,A -85,B 0,C 180,E1 -457.633,E2 -457.633} C_VEL
LIN {X 0,Y 608.497,Z 738.723,A -85,B 0,C 180,E1 -458.134,E2 -458.134} C_VEL
LIN {X 0,Y 608.501,Z 730.393,A -85,B 0,C 180,E1 -458.551,E2 -458.551} C_VEL
LIN {X 0,Y 608.49,Z 721.895,A -85,B 0,C 180,E1 -458.886,E2 -458.886} C_VEL
LIN {X 0,Y 608.509,Z 712.594,A -85,B 0,C 180,E1 -459.158,E2 -459.158} C_VEL
LIN {X 0,Y 608.503,Z 701.563,A -85,B 0,C 180,E1 -459.368,E2 -459.368} C_VEL
LIN {X 0,Y 608.519,Z 627.165,A -85,B 0,C 180,E1 -460.249,E2 -460.249} C_VEL
LIN {X 0,Y 608.466,Z 626.142,A -85,B 0,C 180,E1 -460.313,E2 -460.313} C_VEL
LIN {X 0,Y 608.488,Z 604.917,A -85,B 0,C 180,E1 -463.016,E2 -463.016} C_VEL
LIN {X 0,Y 608.488,Z 583.735,A -85,B 0,C 180,E1 -465.749,E2 -465.749} C_VEL
LIN {X 0,Y 608.53,Z 562.716,A -85,B 0,C 180,E1 -468.496,E2 -468.496} C_VEL
LIN {X 0,Y 608.571,Z 542.695,A -85,B 0,C 180,E1 -471.154,E2 -471.154} C_VEL
LIN {X 0,Y 608.606,Z 522.837,A -85,B 0,C 180,E1 -473.838,E2 -473.838} C_VEL
LIN {X 0,Y 608.658,Z 502.979,A -85,B 0,C 180,E1 -476.579,E2 -476.579} C_VEL
LIN {X 0,Y 608.498,Z 499.663,A -85,B 0,C 180,E1 -477.077,E2 -477.077} C_VEL
LIN {X 0,Y 608.465,Z 499.498,A -85,B 0,C 180,E1 -479.971,E2 -479.971} C_VEL
LIN {X 0,Y 608.457,Z 499.502,A -85,B 0,C 180,E1 -482.522,E2 -482.522} C_VEL
LIN {X 0,Y 608.434,Z 499.507,A -85,B 0,C 180,E1 -485.277,E2 -485.277} C_VEL
LIN {X 0,Y 608.47,Z 499.498,A -85,B 0,C 180,E1 -487.745,E2 -487.745} C_VEL
LIN {X 0,Y 608.45,Z 499.501,A -85,B 0,C 180,E1 -490.329,E2 -490.329} C_VEL
LIN {X 0,Y 608.484,Z 499.5,A -85,B 0,C 180,E1 -493.31,E2 -493.31} C_VEL
LIN {X 0,Y 608.466,Z 499.498,A -85,B 0,C 180,E1 -496.13,E2 -496.13} C_VEL
LIN {X 0,Y 608.458,Z 499.508,A -85,B 0,C 180,E1 -498.824,E2 -498.824} C_VEL
LIN {X 0,Y 608.471,Z 499.5,A -85,B 0,C 180,E1 -501.412,E2 -501.412} C_VEL
LIN {X 0,Y 608.471,Z 499.497,A -85,B 0,C 180,E1 -503.949,E2 -503.949} C_VEL
LIN {X 0,Y 608.461,Z 499.5,A -85,B 0,C 180,E1 -506.329,E2 -506.329} C_VEL
LIN {X 0,Y 608.471,Z 499.505,A -85,B 0,C 180,E1 -508.726,E2 -508.726} C_VEL
LIN {X 0,Y 608.473,Z 499.5,A -85,B 0,C 180,E1 -511.378,E2 -511.378} C_VEL
LIN {X 0,Y 608.449,Z 499.5,A -85,B 0,C 180,E1 -513.965,E2 -513.965} C_VEL
LIN {X 0,Y 608.453,Z 499.51,A -85,B 0,C 180,E1 -516.876,E2 -516.876} C_VEL
LIN {X 0,Y 608.459,Z 499.499,A -85,B 0,C 180,E1 -519.726,E2 -519.726} C_VEL
LIN {X 0,Y 608.446,Z 499.505,A -85,B 0,C 180,E1 -522.523,E2 -522.523} C_VEL
LIN {X 0,Y 608.477,Z 499.501,A -85,B 0,C 180,E1 -525.28,E2 -525.28} C_VEL
LIN {X 0,Y 608.457,Z 499.499,A -85,B 0,C 180,E1 -528,E2 -528} C_VEL
LIN {X 0,Y 608.468,Z 499.506,A -85,B 0,C 180,E1 -530.694,E2 -530.694} C_VEL
LIN {X 0,Y 608.465,Z 499.501,A -85,B 0,C 180,E1 -533.368,E2 -533.368} C_VEL
LIN {X 0,Y 608.446,Z 499.501,A -85,B 0,C 180,E1 -536.026,E2 -536.026} C_VEL
LIN {X 0,Y 608.47,Z 499.505,A -85,B 0,C 180,E1 -538.677,E2 -538.677} C_VEL
LIN {X 0,Y 608.473,Z 499.5,A -85,B 0,C 180,E1 -541.324,E2 -541.324} C_VEL
LIN {X 0,Y 608.448,Z 499.5,A -85,B 0,C 180,E1 -543.974,E2 -543.974} C_VEL
LIN {X 0,Y 608.466,Z 499.506,A -85,B 0,C 180,E1 -546.633,E2 -546.633} C_VEL
LIN {X 0,Y 608.459,Z 499.504,A -85,B 0,C 180,E1 -548.474,E2 -548.474} C_VEL
LIN {X 0,Y 608.102,Z 500.113,A -85,B 0,C 180,E1 -548.638,E2 -548.638} C_VEL
LIN {X 0,Y 606.772,Z 502.418,A -85,B 0,C 180,E1 -548.811,E2 -548.811} C_VEL
LIN {X 0,Y 604.424,Z 506.931,A -85,B 0,C 180,E1 -548.902,E2 -548.902} C_VEL
LIN {X 0,Y 602.492,Z 512.921,A -85,B 0,C 180,E1 -548.929,E2 -548.929} C_VEL
LIN {X 0,Y 601.704,Z 519.988,A -85,B 0,C 180,E1 -548.993,E2 -548.993} C_VEL
LIN {X 0,Y 601.623,Z 529.491,A -85,B 0,C 180,E1 -549.119,E2 -549.119} C_VEL
LIN {X 0,Y 601.598,Z 542.95,A -85,B 0,C 180,E1 -549.371,E2 -549.371} C_VEL
LIN {X 0,Y 601.547,Z 555.785,A -85,B 0,C 180,E1 -549.754,E2 -549.754} C_VEL
LIN {X 0,Y 601.515,Z 568.044,A -85,B 0,C 180,E1 -550.264,E2 -550.264} C_VEL
LIN {X 0,Y 601.49,Z 580.393,A -85,B 0,C 180,E1 -550.939,E2 -550.939} C_VEL
LIN {X 0,Y 601.446,Z 591.467,A -85,B 0,C 180,E1 -551.714,E2 -551.714} C_VEL
LIN {X 0,Y 601.418,Z 600.426,A -85,B 0,C 180,E1 -552.485,E2 -552.485} C_VEL
LIN {X 0,Y 601.391,Z 608.679,A -85,B 0,C 180,E1 -553.345,E2 -553.345} C_VEL
LIN {X 0,Y 601.39,Z 616.793,A -85,B 0,C 180,E1 -554.379,E2 -554.379} C_VEL
LIN {X 0,Y 601.375,Z 622.297,A -85,B 0,C 180,E1 -555.245,E2 -555.245} C_VEL
LIN {X 0,Y 601.362,Z 627.67,A -85,B 0,C 180,E1 -556.289,E2 -556.289} C_VEL
LIN {X 0,Y 601.34,Z 631.822,A -85,B 0,C 180,E1 -557.339,E2 -557.339} C_VEL
LIN {X 0,Y 601.321,Z 634.872,A -85,B 0,C 180,E1 -558.395,E2 -558.395} C_VEL
LIN {X 0,Y 601.321,Z 636.312,A -85,B 0,C 180,E1 -559.102,E2 -559.102} C_VEL
LIN {X 0,Y 601.314,Z 637.307,A -85,B 0,C 180,E1 -559.813,E2 -559.813} C_VEL
LIN {X 0,Y 601.334,Z 637.944,A -85,B 0,C 180,E1 -560.778,E2 -560.778} C_VEL
LIN {X 0,Y 601.333,Z 637.612,A -85,B 0,C 180,E1 -561.963,E2 -561.963} C_VEL
LIN {X 0,Y 601.311,Z 636.801,A -85,B 0,C 180,E1 -562.687,E2 -562.687} C_VEL
LIN {X 0,Y 601.319,Z 635.487,A -85,B 0,C 180,E1 -563.415,E2 -563.415} C_VEL
LIN {X 0,Y 601.329,Z 633.338,A -85,B 0,C 180,E1 -564.273,E2 -564.273} C_VEL
LIN {X 0,Y 601.37,Z 629.996,A -85,B 0,C 180,E1 -565.25,E2 -565.25} C_VEL
LIN {X 0,Y 601.379,Z 624.908,A -85,B 0,C 180,E1 -566.365,E2 -566.365} C_VEL
LIN {X 0,Y 601.361,Z 619.158,A -85,B 0,C 180,E1 -567.355,E2 -567.355} C_VEL
LIN {X 0,Y 601.407,Z 611.264,A -85,B 0,C 180,E1 -568.438,E2 -568.438} C_VEL
LIN {X 0,Y 601.424,Z 602.639,A -85,B 0,C 180,E1 -569.393,E2 -569.393} C_VEL
LIN {X 0,Y 601.45,Z 592.922,A -85,B 0,C 180,E1 -570.26,E2 -570.26} C_VEL
LIN {X 0,Y 601.495,Z 582.399,A -85,B 0,C 180,E1 -571.022,E2 -571.022} C_VEL
LIN {X 0,Y 601.532,Z 571.791,A -85,B 0,C 180,E1 -571.639,E2 -571.639} C_VEL
LIN {X 0,Y 601.538,Z 560.38,A -85,B 0,C 180,E1 -572.163,E2 -572.163} C_VEL
LIN {X 0,Y 601.585,Z 547.25,A -85,B 0,C 180,E1 -572.606,E2 -572.606} C_VEL
LIN {X 0,Y 601.615,Z 534.11,A -85,B 0,C 180,E1 -572.903,E2 -572.903} C_VEL
LIN {X 0,Y 601.599,Z 501.357,A -85,B 0,C 180,E1 -573.328,E2 -573.328} C_VEL
LIN {X 0,Y 601.44,Z 500.431,A -85,B 0,C 180,E1 -573.463,E2 -573.463} C_VEL
LIN {X 0,Y 601.439,Z 500.374,A -85,B 0,C 180,E1 -576.267,E2 -576.267} C_VEL
LIN {X 0,Y 601.432,Z 500.382,A -85,B 0,C 180,E1 -579.125,E2 -579.125} C_VEL
LIN {X 0,Y 601.421,Z 500.379,A -85,B 0,C 180,E1 -581.766,E2 -581.766} C_VEL
LIN {X 0,Y 601.421,Z 500.376,A -85,B 0,C 180,E1 -584.536,E2 -584.536} C_VEL
LIN {X 0,Y 601.437,Z 500.384,A -85,B 0,C 180,E1 -587.407,E2 -587.407} C_VEL
LIN {X 0,Y 601.436,Z 500.373,A -85,B 0,C 180,E1 -590.465,E2 -590.465} C_VEL
LIN {X 0,Y 601.403,Z 500.389,A -85,B 0,C 180,E1 -593.418,E2 -593.418} C_VEL
LIN {X 0,Y 601.432,Z 500.376,A -85,B 0,C 180,E1 -596.065,E2 -596.065} C_VEL
LIN {X 0,Y 601.431,Z 500.374,A -85,B 0,C 180,E1 -598.545,E2 -598.545} C_VEL
LIN {X 0,Y 601.436,Z 500.382,A -85,B 0,C 180,E1 -601.374,E2 -601.374} C_VEL
LIN {X 0,Y 601.405,Z 500.386,A -85,B 0,C 180,E1 -603.637,E2 -603.637} C_VEL
LIN {X 0,Y 601.463,Z 500.375,A -85,B 0,C 180,E1 -605.861,E2 -605.861} C_VEL
LIN {X 0,Y 601.406,Z 500.377,A -85,B 0,C 180,E1 -608.761,E2 -608.761} C_VEL
LIN {X 0,Y 601.421,Z 500.386,A -85,B 0,C 180,E1 -611.609,E2 -611.609} C_VEL
LIN {X 0,Y 601.417,Z 500.376,A -85,B 0,C 180,E1 -614.409,E2 -614.409} C_VEL
LIN {X 0,Y 601.419,Z 500.379,A -85,B 0,C 180,E1 -617.172,E2 -617.172} C_VEL
LIN {X 0,Y 601.432,Z 500.38,A -85,B 0,C 180,E1 -619.905,E2 -619.905} C_VEL
LIN {X 0,Y 601.444,Z 500.372,A -85,B 0,C 180,E1 -622.615,E2 -622.615} C_VEL
LIN {X 0,Y 601.418,Z 500.38,A -85,B 0,C 180,E1 -625.308,E2 -625.308} C_VEL
LIN {X 0,Y 601.434,Z 500.38,A -85,B 0,C 180,E1 -627.991,E2 -627.991} C_VEL
LIN {X 0,Y 601.444,Z 500.372,A -85,B 0,C 180,E1 -630.67,E2 -630.67} C_VEL
LIN {X 0,Y 601.429,Z 500.378,A -85,B 0,C 180,E1 -633.35,E2 -633.35} C_VEL
LIN {X 0,Y 601.42,Z 500.382,A -85,B 0,C 180,E1 -636.037,E2 -636.037} C_VEL
LIN {X 0,Y 601.411,Z 500.376,A -85,B 0,C 180,E1 -638.738,E2 -638.738} C_VEL
LIN {X 0,Y 601.439,Z 500.377,A -85,B 0,C 180,E1 -641.458,E2 -641.458} C_VEL
LIN {X 0,Y 601.424,Z 500.38,A -85,B 0,C 180,E1 -644.205,E2 -644.205} C_VEL
LIN {X 0,Y 601.416,Z 500.376,A -85,B 0,C 180,E1 -646.986,E2 -646.986} C_VEL
LIN {X 0,Y 601.409,Z 500.386,A -85,B 0,C 180,E1 -649.809,E2 -649.809} C_VEL
LIN {X 0,Y 601.414,Z 500.377,A -85,B 0,C 180,E1 -652.682,E2 -652.682} C_VEL
LIN {X 0,Y 601.403,Z 500.378,A -85,B 0,C 180,E1 -654.878,E2 -654.878} C_VEL
LIN {X 0,Y 601.421,Z 500.385,A -85,B 0,C 180,E1 -657.867,E2 -657.867} C_VEL
LIN {X 0,Y 601.43,Z 500.382,A -85,B 0,C 180,E1 -660.163,E2 -660.163} C_VEL
LIN {X 0,Y 601.419,Z 500.376,A -85,B 0,C 180,E1 -662.714,E2 -662.714} C_VEL
LIN {X 0,Y 601.391,Z 500.379,A -85,B 0,C 180,E1 -665.111,E2 -665.111} C_VEL
LIN {X 0,Y 601.436,Z 500.375,A -85,B 0,C 180,E1 -667.418,E2 -667.418} C_VEL
LIN {X 0,Y 601.411,Z 500.386,A -85,B 0,C 180,E1 -669.994,E2 -669.994} C_VEL
LIN {X 0,Y 601.412,Z 500.378,A -85,B 0,C 180,E1 -672.669,E2 -672.669} C_VEL
LIN {X 0,Y 601.423,Z 500.376,A -85,B 0,C 180,E1 -675.481,E2 -675.481} C_VEL
LIN {X 0,Y 601.42,Z 500.382,A -85,B 0,C 180,E1 -678.406,E2 -678.406} C_VEL
LIN {X 0,Y 601.432,Z 500.375,A -85,B 0,C 180,E1 -680.875,E2 -680.875} C_VEL
LIN {X 0,Y 601.439,Z 500.376,A -85,B 0,C 180,E1 -683.733,E2 -683.733} C_VEL
LIN {X 0,Y 601.43,Z 500.383,A -85,B 0,C 180,E1 -686.063,E2 -686.063} C_VEL
LIN {X 0,Y 601.436,Z 500.379,A -85,B 0,C 180,E1 -688.541,E2 -688.541} C_VEL
LIN {X 0,Y 601.43,Z 500.374,A -85,B 0,C 180,E1 -691.373,E2 -691.373} C_VEL
LIN {X 0,Y 601.419,Z 500.384,A -85,B 0,C 180,E1 -694.129,E2 -694.129} C_VEL
LIN {X 0,Y 601.417,Z 500.381,A -85,B 0,C 180,E1 -696.589,E2 -696.589} C_VEL
LIN {X 0,Y 601.428,Z 500.375,A -85,B 0,C 180,E1 -699.478,E2 -699.478} C_VEL
LIN {X 0,Y 601.392,Z 500.39,A -85,B 0,C 180,E1 -702.311,E2 -702.311} C_VEL
LIN {X 0,Y 601.409,Z 500.387,A -85,B 0,C 180,E1 -704.408,E2 -704.408} C_VEL
LIN {X 0,Y 601.419,Z 500.376,A -85,B 0,C 180,E1 -707.172,E2 -707.172} C_VEL
LIN {X 0,Y 601.428,Z 500.377,A -85,B 0,C 180,E1 -709.905,E2 -709.905} C_VEL
LIN {X 0,Y 601.445,Z 500.38,A -85,B 0,C 180,E1 -712.615,E2 -712.615} C_VEL
LIN {X 0,Y 601.429,Z 500.374,A -85,B 0,C 180,E1 -715.308,E2 -715.308} C_VEL
LIN {X 0,Y 601.418,Z 500.379,A -85,B 0,C 180,E1 -717.991,E2 -717.991} C_VEL
LIN {X 0,Y 601.448,Z 500.38,A -85,B 0,C 180,E1 -720.669,E2 -720.669} C_VEL
LIN {X 0,Y 601.426,Z 500.375,A -85,B 0,C 180,E1 -723.349,E2 -723.349} C_VEL
LIN {X 0,Y 601.406,Z 500.38,A -85,B 0,C 180,E1 -726.037,E2 -726.037} C_VEL
LIN {X 0,Y 601.434,Z 500.381,A -85,B 0,C 180,E1 -728.737,E2 -728.737} C_VEL
LIN {X 0,Y 601.426,Z 500.375,A -85,B 0,C 180,E1 -731.458,E2 -731.458} C_VEL
LIN {X 0,Y 601.41,Z 500.381,A -85,B 0,C 180,E1 -734.205,E2 -734.205} C_VEL
LIN {X 0,Y 601.426,Z 500.379,A -85,B 0,C 180,E1 -736.986,E2 -736.986} C_VEL
LIN {X 0,Y 601.4,Z 500.378,A -85,B 0,C 180,E1 -739.809,E2 -739.809} C_VEL
LIN {X 0,Y 601.406,Z 500.387,A -85,B 0,C 180,E1 -742.606,E2 -742.606} C_VEL
LIN {X 0,Y 601.398,Z 500.386,A -85,B 0,C 180,E1 -744.879,E2 -744.879} C_VEL
LIN {X 0,Y 601.415,Z 500.376,A -85,B 0,C 180,E1 -747.867,E2 -747.867} C_VEL
LIN {X 0,Y 601.44,Z 500.375,A -85,B 0,C 180,E1 -750.163,E2 -750.163} C_VEL
LIN {X 0,Y 601.417,Z 500.386,A -85,B 0,C 180,E1 -752.717,E2 -752.717} C_VEL
LIN {X 0,Y 601.417,Z 500.381,A -85,B 0,C 180,E1 -755.117,E2 -755.117} C_VEL
LIN {X 0,Y 601.428,Z 500.376,A -85,B 0,C 180,E1 -757.419,E2 -757.419} C_VEL
LIN {X 0,Y 601.406,Z 500.377,A -85,B 0,C 180,E1 -759.995,E2 -759.995} C_VEL
LIN {X 0,Y 601.405,Z 500.385,A -85,B 0,C 180,E1 -762.671,E2 -762.671} C_VEL
LIN {X 0,Y 601.42,Z 500.377,A -85,B 0,C 180,E1 -765.483,E2 -765.483} C_VEL
LIN {X 0,Y 601.422,Z 500.378,A -85,B 0,C 180,E1 -768.407,E2 -768.407} C_VEL
LIN {X 0,Y 601.434,Z 500.384,A -85,B 0,C 180,E1 -770.876,E2 -770.876} C_VEL
LIN {X 0,Y 601.439,Z 500.374,A -85,B 0,C 180,E1 -773.734,E2 -773.734} C_VEL
LIN {X 0,Y 601.423,Z 500.381,A -85,B 0,C 180,E1 -776.687,E2 -776.687} C_VEL
LIN {X 0,Y 601.43,Z 500.385,A -85,B 0,C 180,E1 -779.059,E2 -779.059} C_VEL
LIN {X 0,Y 601.427,Z 500.383,A -85,B 0,C 180,E1 -781.374,E2 -781.374} C_VEL
LIN {X 0,Y 601.446,Z 500.533,A -85,B 0,C 180,E1 -782.702,E2 -782.702} C_VEL
LIN {X 0,Y 601.837,Z 504.302,A -85,B 0,C 180,E1 -783.283,E2 -783.283} C_VEL
LIN {X 0,Y 601.73,Z 522.836,A -85,B 0,C 180,E1 -785.872,E2 -785.872} C_VEL
LIN {X 0,Y 601.653,Z 542.694,A -85,B 0,C 180,E1 -788.591,E2 -788.591} C_VEL
LIN {X 0,Y 601.567,Z 563.429,A -85,B 0,C 180,E1 -791.377,E2 -791.377} C_VEL
LIN {X 0,Y 601.503,Z 583.734,A -85,B 0,C 180,E1 -794.064,E2 -794.064} C_VEL
LIN {X 0,Y 601.461,Z 604.916,A -85,B 0,C 180,E1 -796.829,E2 -796.829} C_VEL
LIN {X 0,Y 601.429,Z 626.144,A -85,B 0,C 180,E1 -799.565,E2 -799.565} C_VEL
LIN {X 0,Y 601.481,Z 627.184,A -85,B 0,C 180,E1 -799.63,E2 -799.63} C_VEL
LIN {X 0,Y 601.517,Z 705.454,A -85,B 0,C 180,E1 -800.586,E2 -800.586} C_VEL
LIN {X 0,Y 601.507,Z 715.913,A -85,B 0,C 180,E1 -800.819,E2 -800.819} C_VEL
LIN {X 0,Y 601.472,Z 726.621,A -85,B 0,C 180,E1 -801.178,E2 -801.178} C_VEL
LIN {X 0,Y 601.447,Z 737.237,A -85,B 0,C 180,E1 -801.686,E2 -801.686} C_VEL
LIN {X 0,Y 601.411,Z 745.546,A -85,B 0,C 180,E1 -802.192,E2 -802.192} C_VEL
LIN {X 0,Y 601.412,Z 753.404,A -85,B 0,C 180,E1 -802.783,E2 -802.783} C_VEL
LIN {X 0,Y 601.411,Z 760.598,A -85,B 0,C 180,E1 -803.443,E2 -803.443} C_VEL
LIN {X 0,Y 601.391,Z 768.191,A -85,B 0,C 180,E1 -804.299,E2 -804.299} C_VEL
LIN {X 0,Y 601.381,Z 774.028,A -85,B 0,C 180,E1 -805.14,E2 -805.14} C_VEL
LIN {X 0,Y 601.343,Z 778.631,A -85,B 0,C 180,E1 -805.979,E2 -805.979} C_VEL
LIN {X 0,Y 601.344,Z 781.622,A -85,B 0,C 180,E1 -806.65,E2 -806.65} C_VEL
LIN {X 0,Y 601.328,Z 783.932,A -85,B 0,C 180,E1 -807.32,E2 -807.32} C_VEL
LIN {X 0,Y 601.34,Z 785.679,A -85,B 0,C 180,E1 -807.991,E2 -807.991} C_VEL
LIN {X 0,Y 601.346,Z 786.934,A -85,B 0,C 180,E1 -808.661,E2 -808.661} C_VEL
LIN {X 0,Y 601.337,Z 787.714,A -85,B 0,C 180,E1 -809.33,E2 -809.33} C_VEL
LIN {X 0,Y 601.332,Z 788,A -85,B 0,C 180,E1 -810,E2 -810} C_VEL
LIN {X 0,Y 601.337,Z 787.714,A -85,B 0,C 180,E1 -810.67,E2 -810.67} C_VEL
LIN {X 0,Y 601.346,Z 786.934,A -85,B 0,C 180,E1 -811.339,E2 -811.339} C_VEL
LIN {X 0,Y 601.34,Z 785.679,A -85,B 0,C 180,E1 -812.009,E2 -812.009} C_VEL
LIN {X 0,Y 601.346,Z 782.787,A -85,B 0,C 180,E1 -813.015,E2 -813.015} C_VEL
LIN {X 0,Y 601.364,Z 780.147,A -85,B 0,C 180,E1 -813.685,E2 -813.685} C_VEL
LIN {X 0,Y 601.367,Z 774.986,A -85,B 0,C 180,E1 -814.692,E2 -814.692} C_VEL
LIN {X 0,Y 601.383,Z 769.432,A -85,B 0,C 180,E1 -815.532,E2 -815.532} C_VEL
LIN {X 0,Y 601.393,Z 762.152,A -85,B 0,C 180,E1 -816.403,E2 -816.403} C_VEL
LIN {X 0,Y 601.415,Z 754.418,A -85,B 0,C 180,E1 -817.132,E2 -817.132} C_VEL
LIN {X 0,Y 601.431,Z 746.765,A -85,B 0,C 180,E1 -817.723,E2 -817.723} C_VEL
LIN {X 0,Y 601.455,Z 738.725,A -85,B 0,C 180,E1 -818.229,E2 -818.229} C_VEL
LIN {X 0,Y 601.481,Z 730.396,A -85,B 0,C 180,E1 -818.652,E2 -818.652} C_VEL
LIN {X 0,Y 601.471,Z 721.896,A -85,B 0,C 180,E1 -818.991,E2 -818.991} C_VEL
LIN {X 0,Y 601.493,Z 712.595,A -85,B 0,C 180,E1 -819.266,E2 -819.266} C_VEL
LIN {X 0,Y 601.525,Z 701.563,A -85,B 0,C 180,E1 -819.478,E2 -819.478} C_VEL
LIN {X 0,Y 601.481,Z 627.154,A -85,B 0,C 180,E1 -820.37,E2 -820.37} C_VEL
LIN {X 0,Y 601.429,Z 626.142,A -85,B 0,C 180,E1 -820.435,E2 -820.435} C_VEL
LIN {X 0,Y 601.461,Z 604.917,A -85,B 0,C 180,E1 -823.17,E2 -823.17} C_VEL
LIN {X 0,Y 601.503,Z 583.735,A -85,B 0,C 180,E1 -825.936,E2 -825.936} C_VEL
LIN {X 0,Y 601.587,Z 563.431,A -85,B 0,C 180,E1 -828.622,E2 -828.622} C_VEL
LIN {X 0,Y 601.653,Z 542.695,A -85,B 0,C 180,E1 -831.409,E2 -831.409} C_VEL
LIN {X 0,Y 601.741,Z 522.837,A -85,B 0,C 180,E1 -834.128,E2 -834.128} C_VEL
LIN {X 0,Y 601.867,Z 502.979,A -85,B 0,C 180,E1 -836.902,E2 -836.902} C_VEL
LIN {X 0,Y 601.462,Z 500.469,A -85,B 0,C 180,E1 -837.33,E2 -837.33} C_VEL
LIN {X 0,Y 601.426,Z 500.376,A -85,B 0,C 180,E1 -840.163,E2 -840.163} C_VEL
LIN {X 0,Y 601.419,Z 500.382,A -85,B 0,C 180,E1 -842.715,E2 -842.715} C_VEL
LIN {X 0,Y 601.391,Z 500.388,A -85,B 0,C 180,E1 -845.111,E2 -845.111} C_VEL
LIN {X 0,Y 601.433,Z 500.378,A -85,B 0,C 180,E1 -847.418,E2 -847.418} C_VEL
LIN {X 0,Y 601.409,Z 500.377,A -85,B 0,C 180,E1 -849.994,E2 -849.994} C_VEL
LIN {X 0,Y 601.435,Z 500.38,A -85,B 0,C 180,E1 -852.667,E2 -852.667} C_VEL
LIN {X 0,Y 601.419,Z 500.378,A -85,B 0,C 180,E1 -855.481,E2 -855.481} C_VEL
LIN {X 0,Y 601.42,Z 500.378,A -85,B 0,C 180,E1 -858.406,E2 -858.406} C_VEL
LIN {X 0,Y 601.437,Z 500.384,A -85,B 0,C 180,E1 -860.876,E2 -860.876} C_VEL
LIN {X 0,Y 601.439,Z 500.374,A -85,B 0,C 180,E1 -863.733,E2 -863.733} C_VEL
LIN {X 0,Y 601.429,Z 500.375,A -85,B 0,C 180,E1 -866.063,E2 -866.063} C_VEL
LIN {X 0,Y 601.435,Z 500.378,A -85,B 0,C 180,E1 -868.541,E2 -868.541} C_VEL
LIN {X 0,Y 601.432,Z 500.378,A -85,B 0,C 180,E1 -871.373,E2 -871.373} C_VEL
LIN {X 0,Y 601.405,Z 500.378,A -85,B 0,C 180,E1 -873.637,E2 -873.637} C_VEL
LIN {X 0,Y 601.419,Z 500.381,A -85,B 0,C 180,E1 -876.59,E2 -876.59} C_VEL
LIN {X 0,Y 601.429,Z 500.376,A -85,B 0,C 180,E1 -879.478,E2 -879.478} C_VEL
LIN {X 0,Y 601.392,Z 500.381,A -85,B 0,C 180,E1 -882.312,E2 -882.312} C_VEL
LIN {X 0,Y 601.415,Z 500.38,A -85,B 0,C 180,E1 -884.409,E2 -884.409} C_VEL
LIN {X 0,Y 601.422,Z 500.381,A -85,B 0,C 180,E1 -887.172,E2 -887.172} C_VEL
LIN {X 0,Y 601.429,Z 500.375,A -85,B 0,C 180,E1 -889.905,E2 -889.905} C_VEL
LIN {X 0,Y 601.45,Z 500.379,A -85,B 0,C 180,E1 -892.615,E2 -892.615} C_VEL
LIN {X 0,Y 601.431,Z 500.378,A -85,B 0,C 180,E1 -895.308,E2 -895.308} C_VEL
LIN {X 0,Y 601.418,Z 500.376,A -85,B 0,C 180,E1 -897.991,E2 -897.991} C_VEL
LIN {X 0,Y 601.453,Z 500.38,A -85,B 0,C 180,E1 -900.67,E2 -900.67} C_VEL
LIN {X 0,Y 601.432,Z 500.377,A -85,B 0,C 180,E1 -903.35,E2 -903.35} C_VEL
LIN {X 0,Y 601.426,Z 500.376,A -85,B 0,C 180,E1 -906.037,E2 -906.037} C_VEL
LIN {X 0,Y 601.454,Z 500.577,A -85,B 0,C 180,E1 -908.674,E2 -908.674} C_VEL
LIN {X 0,Y 601.639,Z 501.674,A -85,B 0,C 180,E1 -908.777,E2 -908.777} C_VEL
LIN {X 0,Y 601.623,Z 529.491,A -85,B 0,C 180,E1 -909.119,E2 -909.119} C_VEL
LIN {X 0,Y 601.242,Z 533.385,A -85,B 0,C 180,E1 -909.167,E2 -909.167} C_VEL
LIN {X 0,Y 599.27,Z 540.977,A -85,B 0,C 180,E1 -909.278,E2 -909.278} C_VEL
LIN {X 0,Y 595.351,Z 552.959,A -85,B 0,C 180,E1 -909.537,E2 -909.537} C_VEL
LIN {X 0,Y 594.635,Z 557.586,A -85,B 0,C 180,E1 -909.688,E2 -909.688} C_VEL
LIN {X 0,Y 594.58,Z 559.393,A -85,B 0,C 180,E1 -909.756,E2 -909.756} C_VEL
LIN {X 0,Y 594.539,Z 571.325,A -85,B 0,C 180,E1 -910.3,E2 -910.3} C_VEL
LIN {X 0,Y 594.501,Z 582.593,A -85,B 0,C 180,E1 -910.964,E2 -910.964} C_VEL
LIN {X 0,Y 594.406,Z 593.509,A -85,B 0,C 180,E1 -911.769,E2 -911.769} C_VEL
LIN {X 0,Y 594.369,Z 603.024,A -85,B 0,C 180,E1 -912.636,E2 -912.636} C_VEL
LIN {X 0,Y 594.304,Z 612.211,A -85,B 0,C 180,E1 -913.681,E2 -913.681} C_VEL
LIN {X 0,Y 594.326,Z 619.594,A -85,B 0,C 180,E1 -914.729,E2 -914.729} C_VEL
LIN {X 0,Y 594.279,Z 625.538,A -85,B 0,C 180,E1 -915.784,E2 -915.784} C_VEL
LIN {X 0,Y 594.249,Z 629.525,A -85,B 0,C 180,E1 -916.677,E2 -916.677} C_VEL
LIN {X 0,Y 594.218,Z 633.711,A -85,B 0,C 180,E1 -917.91,E2 -917.91} C_VEL
LIN {X 0,Y 594.239,Z 635.995,A -85,B 0,C 180,E1 -918.892,E2 -918.892} C_VEL
LIN {X 0,Y 594.217,Z 637.573,A -85,B 0,C 180,E1 -920.06,E2 -920.06} C_VEL
LIN {X 0,Y 594.243,Z 637.969,A -85,B 0,C 180,E1 -920.885,E2 -920.885} C_VEL
LIN {X 0,Y 594.244,Z 637.369,A -85,B 0,C 180,E1 -922.238,E2 -922.238} C_VEL
LIN {X 0,Y 594.204,Z 636.373,A -85,B 0,C 180,E1 -922.974,E2 -922.974} C_VEL
LIN {X 0,Y 594.223,Z 634.917,A -85,B 0,C 180,E1 -923.711,E2 -923.711} C_VEL
LIN {X 0,Y 594.261,Z 631.712,A -85,B 0,C 180,E1 -924.825,E2 -924.825} C_VEL
LIN {X 0,Y 594.278,Z 626.986,A -85,B 0,C 180,E1 -926.004,E2 -926.004} C_VEL
LIN {X 0,Y 594.279,Z 620.151,A -85,B 0,C 180,E1 -927.275,E2 -927.275} C_VEL
LIN {X 0,Y 594.32,Z 613.594,A -85,B 0,C 180,E1 -928.23,E2 -928.23} C_VEL
LIN {X 0,Y 594.377,Z 605.485,A -85,B 0,C 180,E1 -929.193,E2 -929.193} C_VEL
LIN {X 0,Y 594.419,Z 595.792,A -85,B 0,C 180,E1 -930.128,E2 -930.128} C_VEL
LIN {X 0,Y 594.455,Z 585.251,A -85,B 0,C 180,E1 -930.95,E2 -930.95} C_VEL
LIN {X 0,Y 594.511,Z 573.636,A -85,B 0,C 180,E1 -931.666,E2 -931.666} C_VEL
LIN {X 0,Y 594.562,Z 561.772,A -85,B 0,C 180,E1 -932.236,E2 -932.236} C_VEL
LIN {X 0,Y 594.635,Z 549.352,A -85,B 0,C 180,E1 -932.683,E2 -932.683} C_VEL
LIN {X 0,Y 594.68,Z 535.226,A -85,B 0,C 180,E1 -933.022,E2 -933.022} C_VEL
LIN {X 0,Y 594.654,Z 502.504,A -85,B 0,C 180,E1 -933.451,E2 -933.451} C_VEL
LIN {X 0,Y 594.41,Z 501.362,A -85,B 0,C 180,E1 -933.578,E2 -933.578} C_VEL
LIN {X 0,Y 594.389,Z 501.253,A -85,B 0,C 180,E1 -936.486,E2 -936.486} C_VEL
LIN {X 0,Y 594.382,Z 501.255,A -85,B 0,C 180,E1 -938.806,E2 -938.806} C_VEL
LIN {X 0,Y 594.38,Z 501.255,A -85,B 0,C 180,E1 -941.85,E2 -941.85} C_VEL
LIN {X 0,Y 594.378,Z 501.253,A -85,B 0,C 180,E1 -944.237,E2 -944.237} C_VEL
LIN {X 0,Y 594.382,Z 501.259,A -85,B 0,C 180,E1 -947.147,E2 -947.147} C_VEL
LIN {X 0,Y 594.388,Z 501.262,A -85,B 0,C 180,E1 -949.436,E2 -949.436} C_VEL
LIN {X 0,Y 594.39,Z 501.251,A -85,B 0,C 180,E1 -952.392,E2 -952.392} C_VEL
LIN {X 0,Y 594.378,Z 501.263,A -85,B 0,C 180,E1 -955.421,E2 -955.421} C_VEL
LIN {X 0,Y 594.386,Z 501.252,A -85,B 0,C 180,E1 -958.357,E2 -958.357} C_VEL
LIN {X 0,Y 594.385,Z 501.255,A -85,B 0,C 180,E1 -961.043,E2 -961.043} C_VEL
LIN {X 0,Y 594.384,Z 501.255,A -85,B 0,C 180,E1 -963.979,E2 -963.979} C_VEL
LIN {X 0,Y 594.38,Z 501.253,A -85,B 0,C 180,E1 -966.296,E2 -966.296} C_VEL
LIN {X 0,Y 594.405,Z 501.254,A -85,B 0,C 180,E1 -969.225,E2 -969.225} C_VEL
LIN {X 0,Y 594.355,Z 501.258,A -85,B 0,C 180,E1 -972.096,E2 -972.096} C_VEL
LIN {X 0,Y 594.371,Z 501.255,A -85,B 0,C 180,E1 -974.22,E2 -974.22} C_VEL
LIN {X 0,Y 594.386,Z 501.253,A -85,B 0,C 180,E1 -976.322,E2 -976.322} C_VEL
LIN {X 0,Y 594.378,Z 501.255,A -85,B 0,C 180,E1 -979.095,E2 -979.095} C_VEL
LIN {X 0,Y 594.416,Z 501.256,A -85,B 0,C 180,E1 -981.844,E2 -981.844} C_VEL
LIN {X 0,Y 594.389,Z 501.251,A -85,B 0,C 180,E1 -984.572,E2 -984.572} C_VEL
LIN {X 0,Y 594.404,Z 501.253,A -85,B 0,C 180,E1 -987.289,E2 -987.289} C_VEL
LIN {X 0,Y 594.419,Z 501.254,A -85,B 0,C 180,E1 -990,E2 -990} C_VEL
LIN {X 0,Y 594.403,Z 501.25,A -85,B 0,C 180,E1 -992.711,E2 -992.711} C_VEL
LIN {X 0,Y 594.392,Z 501.256,A -85,B 0,C 180,E1 -995.428,E2 -995.428} C_VEL
LIN {X 0,Y 594.387,Z 501.256,A -85,B 0,C 180,E1 -998.157,E2 -998.157} C_VEL
LIN {X 0,Y 594.391,Z 501.252,A -85,B 0,C 180,E1 -1001.072,E2 -1001.072} C_VEL
LIN {X 0,Y 594.387,Z 501.259,A -85,B 0,C 180,E1 -1003.679,E2 -1003.679} C_VEL
LIN {X 0,Y 594.375,Z 501.253,A -85,B 0,C 180,E1 -1006.711,E2 -1006.711} C_VEL
LIN {X 0,Y 594.37,Z 501.256,A -85,B 0,C 180,E1 -1009.334,E2 -1009.334} C_VEL
LIN {X 0,Y 594.366,Z 501.258,A -85,B 0,C 180,E1 -1011.503,E2 -1011.503} C_VEL
LIN {X 0,Y 594.392,Z 501.254,A -85,B 0,C 180,E1 -1014.445,E2 -1014.445} C_VEL
LIN {X 0,Y 594.386,Z 501.252,A -85,B 0,C 180,E1 -1016.699,E2 -1016.699} C_VEL
LIN {X 0,Y 594.381,Z 501.252,A -85,B 0,C 180,E1 -1018.998,E2 -1018.998} C_VEL
LIN {X 0,Y 594.385,Z 501.256,A -85,B 0,C 180,E1 -1021.643,E2 -1021.643} C_VEL
LIN {X 0,Y 594.378,Z 501.255,A -85,B 0,C 180,E1 -1024.579,E2 -1024.579} C_VEL
LIN {X 0,Y 594.391,Z 501.255,A -85,B 0,C 180,E1 -1027.608,E2 -1027.608} C_VEL
LIN {X 0,Y 594.372,Z 501.256,A -85,B 0,C 180,E1 -1030.566,E2 -1030.566} C_VEL
LIN {X 0,Y 594.379,Z 501.253,A -85,B 0,C 180,E1 -1033.297,E2 -1033.297} C_VEL
LIN {X 0,Y 594.365,Z 501.265,A -85,B 0,C 180,E1 -1036.159,E2 -1036.159} C_VEL
LIN {X 0,Y 594.377,Z 501.257,A -85,B 0,C 180,E1 -1038.535,E2 -1038.535} C_VEL
LIN {X 0,Y 594.384,Z 501.252,A -85,B 0,C 180,E1 -1041.294,E2 -1041.294} C_VEL
LIN {X 0,Y 594.391,Z 501.255,A -85,B 0,C 180,E1 -1043.758,E2 -1043.758} C_VEL
LIN {X 0,Y 594.376,Z 501.264,A -85,B 0,C 180,E1 -1046.238,E2 -1046.238} C_VEL
LIN {X 0,Y 594.385,Z 501.256,A -85,B 0,C 180,E1 -1048.65,E2 -1048.65} C_VEL
LIN {X 0,Y 594.38,Z 501.253,A -85,B 0,C 180,E1 -1051.04,E2 -1051.04} C_VEL
LIN {X 0,Y 594.391,Z 501.257,A -85,B 0,C 180,E1 -1053.974,E2 -1053.974} C_VEL
LIN {X 0,Y 594.386,Z 501.263,A -85,B 0,C 180,E1 -1056.295,E2 -1056.295} C_VEL
LIN {X 0,Y 594.401,Z 501.25,A -85,B 0,C 180,E1 -1059.224,E2 -1059.224} C_VEL
LIN {X 0,Y 594.374,Z 501.26,A -85,B 0,C 180,E1 -1062.095,E2 -1062.095} C_VEL
LIN {X 0,Y 594.362,Z 501.263,A -85,B 0,C 180,E1 -1064.219,E2 -1064.219} C_VEL
LIN {X 0,Y 594.364,Z 501.256,A -85,B 0,C 180,E1 -1067.017,E2 -1067.017} C_VEL
LIN {X 0,Y 594.388,Z 501.253,A -85,B 0,C 180,E1 -1069.784,E2 -1069.784} C_VEL
LIN {X 0,Y 594.393,Z 501.26,A -85,B 0,C 180,E1 -1072.527,E2 -1072.527} C_VEL
LIN {X 0,Y 594.397,Z 501.251,A -85,B 0,C 180,E1 -1075.252,E2 -1075.252} C_VEL
LIN {X 0,Y 594.388,Z 501.254,A -85,B 0,C 180,E1 -1077.967,E2 -1077.967} C_VEL
LIN {X 0,Y 594.419,Z 501.255,A -85,B 0,C 180,E1 -1080.677,E2 -1080.677} C_VEL
LIN {X 0,Y 594.377,Z 501.253,A -85,B 0,C 180,E1 -1083.389,E2 -1083.389} C_VEL
LIN {X 0,Y 594.362,Z 501.258,A -85,B 0,C 180,E1 -1086.109,E2 -1086.109} C_VEL
LIN {X 0,Y 594.394,Z 501.256,A -85,B 0,C 180,E1 -1088.842,E2 -1088.842} C_VEL
LIN {X 0,Y 594.386,Z 501.252,A -85,B 0,C 180,E1 -1091.596,E2 -1091.596} C_VEL
LIN {X 0,Y 594.38,Z 501.259,A -85,B 0,C 180,E1 -1094.377,E2 -1094.377} C_VEL
LIN {X 0,Y 594.383,Z 501.254,A -85,B 0,C 180,E1 -1097.193,E2 -1097.193} C_VEL
LIN {X 0,Y 594.37,Z 501.255,A -85,B 0,C 180,E1 -1100.054,E2 -1100.054} C_VEL
LIN {X 0,Y 594.356,Z 501.261,A -85,B 0,C 180,E1 -1102.967,E2 -1102.967} C_VEL
LIN {X 0,Y 594.374,Z 501.256,A -85,B 0,C 180,E1 -1105.193,E2 -1105.193} C_VEL
LIN {X 0,Y 594.376,Z 501.253,A -85,B 0,C 180,E1 -1107.527,E2 -1107.527} C_VEL
LIN {X 0,Y 594.392,Z 501.255,A -85,B 0,C 180,E1 -1110.331,E2 -1110.331} C_VEL
LIN {X 0,Y 594.371,Z 501.261,A -85,B 0,C 180,E1 -1112.95,E2 -1112.95} C_VEL
LIN {X 0,Y 594.38,Z 501.254,A -85,B 0,C 180,E1 -1115.407,E2 -1115.407} C_VEL
LIN {X 0,Y 594.38,Z 501.253,A -85,B 0,C 180,E1 -1117.941,E2 -1117.941} C_VEL
LIN {X 0,Y 594.372,Z 501.265,A -85,B 0,C 180,E1 -1120.823,E2 -1120.823} C_VEL
LIN {X 0,Y 594.36,Z 501.258,A -85,B 0,C 180,E1 -1123.3,E2 -1123.3} C_VEL
LIN {X 0,Y 594.377,Z 501.254,A -85,B 0,C 180,E1 -1126.159,E2 -1126.159} C_VEL
LIN {X 0,Y 594.376,Z 501.259,A -85,B 0,C 180,E1 -1129.178,E2 -1129.178} C_VEL
LIN {X 0,Y 594.385,Z 501.252,A -85,B 0,C 180,E1 -1132.06,E2 -1132.06} C_VEL
LIN {X 0,Y 594.351,Z 501.263,A -85,B 0,C 180,E1 -1134.676,E2 -1134.676} C_VEL
LIN {X 0,Y 594.376,Z 501.262,A -85,B 0,C 180,E1 -1137.089,E2 -1137.089} C_VEL
LIN {X 0,Y 594.385,Z 501.254,A -85,B 0,C 180,E1 -1139.672,E2 -1139.672} C_VEL
LIN {X 0,Y 594.428,Z 501.473,A -85,B 0,C 180,E1 -1142.495,E2 -1142.495} C_VEL
LIN {X 0,Y 595.009,Z 505.626,A -85,B 0,C 180,E1 -1143.142,E2 -1143.142} C_VEL
LIN {X 0,Y 594.865,Z 524.16,A -85,B 0,C 180,E1 -1145.761,E2 -1145.761} C_VEL
LIN {X 0,Y 594.763,Z 542.695,A -85,B 0,C 180,E1 -1148.33,E2 -1148.33} C_VEL
LIN {X 0,Y 594.608,Z 562.369,A -85,B 0,C 180,E1 -1151.008,E2 -1151.008} C_VEL
LIN {X 0,Y 594.533,Z 582.411,A -85,B 0,C 180,E1 -1153.695,E2 -1153.695} C_VEL
LIN {X 0,Y 594.447,Z 604.916,A -85,B 0,C 180,E1 -1156.671,E2 -1156.671} C_VEL
LIN {X 0,Y 594.37,Z 626.36,A -85,B 0,C 180,E1 -1159.461,E2 -1159.461} C_VEL
LIN {X 0,Y 594.559,Z 628.526,A -85,B 0,C 180,E1 -1159.529,E2 -1159.529} C_VEL
LIN {X 0,Y 594.533,Z 704.154,A -85,B 0,C 180,E1 -1160.453,E2 -1160.453} C_VEL
LIN {X 0,Y 594.507,Z 713.424,A -85,B 0,C 180,E1 -1160.645,E2 -1160.645} C_VEL
LIN {X 0,Y 594.46,Z 721.896,A -85,B 0,C 180,E1 -1160.902,E2 -1160.902} C_VEL
LIN {X 0,Y 594.446,Z 730.396,A -85,B 0,C 180,E1 -1161.245,E2 -1161.245} C_VEL
LIN {X 0,Y 594.431,Z 738.726,A -85,B 0,C 180,E1 -1161.673,E2 -1161.673} C_VEL
LIN {X 0,Y 594.367,Z 746.766,A -85,B 0,C 180,E1 -1162.185,E2 -1162.185} C_VEL
LIN {X 0,Y 594.356,Z 754.418,A -85,B 0,C 180,E1 -1162.783,E2 -1162.783} C_VEL
LIN {X 0,Y 594.33,Z 762.809,A -85,B 0,C 180,E1 -1163.589,E2 -1163.589} C_VEL
LIN {X 0,Y 594.309,Z 769.432,A -85,B 0,C 180,E1 -1164.401,E2 -1164.401} C_VEL
LIN {X 0,Y 594.276,Z 774.986,A -85,B 0,C 180,E1 -1165.252,E2 -1165.252} C_VEL
LIN {X 0,Y 594.285,Z 780.147,A -85,B 0,C 180,E1 -1166.271,E2 -1166.271} C_VEL
LIN {X 0,Y 594.249,Z 782.787,A -85,B 0,C 180,E1 -1166.949,E2 -1166.949} C_VEL
LIN {X 0,Y 594.239,Z 785.679,A -85,B 0,C 180,E1 -1167.967,E2 -1167.967} C_VEL
LIN {X 0,Y 594.246,Z 786.935,A -85,B 0,C 180,E1 -1168.645,E2 -1168.645} C_VEL
LIN {X 0,Y 594.237,Z 787.713,A -85,B 0,C 180,E1 -1169.322,E2 -1169.322} C_VEL
LIN {X 0,Y 594.233,Z 788,A -85,B 0,C 180,E1 -1170,E2 -1170} C_VEL
LIN {X 0,Y 594.237,Z 787.713,A -85,B 0,C 180,E1 -1170.678,E2 -1170.678} C_VEL
LIN {X 0,Y 594.246,Z 786.935,A -85,B 0,C 180,E1 -1171.355,E2 -1171.355} C_VEL
LIN {X 0,Y 594.239,Z 785.68,A -85,B 0,C 180,E1 -1172.033,E2 -1172.033} C_VEL
LIN {X 0,Y 594.249,Z 782.788,A -85,B 0,C 180,E1 -1173.051,E2 -1173.051} C_VEL
LIN {X 0,Y 594.285,Z 780.147,A -85,B 0,C 180,E1 -1173.729,E2 -1173.729} C_VEL
LIN {X 0,Y 594.276,Z 774.987,A -85,B 0,C 180,E1 -1174.748,E2 -1174.748} C_VEL
LIN {X 0,Y 594.309,Z 769.432,A -85,B 0,C 180,E1 -1175.599,E2 -1175.599} C_VEL
LIN {X 0,Y 594.344,Z 762.151,A -85,B 0,C 180,E1 -1176.479,E2 -1176.479} C_VEL
LIN {X 0,Y 594.356,Z 754.419,A -85,B 0,C 180,E1 -1177.217,E2 -1177.217} C_VEL
LIN {X 0,Y 594.367,Z 746.767,A -85,B 0,C 180,E1 -1177.815,E2 -1177.815} C_VEL
LIN {X 0,Y 594.431,Z 738.727,A -85,B 0,C 180,E1 -1178.327,E2 -1178.327} C_VEL
LIN {X 0,Y 594.446,Z 730.399,A -85,B 0,C 180,E1 -1178.755,E2 -1178.755} C_VEL
LIN {X 0,Y 594.459,Z 721.898,A -85,B 0,C 180,E1 -1179.098,E2 -1179.098} C_VEL
LIN {X 0,Y 594.493,Z 711.765,A -85,B 0,C 180,E1 -1179.398,E2 -1179.398} C_VEL
LIN {X 0,Y 594.551,Z 700.081,A -85,B 0,C 180,E1 -1179.611,E2 -1179.611} C_VEL
LIN {X 0,Y 594.428,Z 627.143,A -85,B 0,C 180,E1 -1180.495,E2 -1180.495} C_VEL
LIN {X 0,Y 594.385,Z 626.142,A -85,B 0,C 180,E1 -1180.56,E2 -1180.56} C_VEL
LIN {X 0,Y 594.447,Z 604.917,A -85,B 0,C 180,E1 -1183.329,E2 -1183.329} C_VEL
LIN {X 0,Y 594.535,Z 582.411,A -85,B 0,C 180,E1 -1186.304,E2 -1186.304} C_VEL
LIN {X 0,Y 594.677,Z 559.906,A -85,B 0,C 180,E1 -1189.323,E2 -1189.323} C_VEL
LIN {X 0,Y 594.806,Z 537.613,A -85,B 0,C 180,E1 -1192.369,E2 -1192.369} C_VEL
LIN {X 0,Y 594.918,Z 516.218,A -85,B 0,C 180,E1 -1195.355,E2 -1195.355} C_VEL
LIN {X 0,Y 595.006,Z 504.303,A -85,B 0,C 180,E1 -1197.048,E2 -1197.048} C_VEL
LIN {X 0,Y 594.402,Z 501.394,A -85,B 0,C 180,E1 -1197.53,E2 -1197.53} C_VEL
LIN {X 0,Y 594.385,Z 501.254,A -85,B 0,C 180,E1 -1200.328,E2 -1200.328} C_VEL
LIN {X 0,Y 594.375,Z 501.264,A -85,B 0,C 180,E1 -1202.949,E2 -1202.949} C_VEL
LIN {X 0,Y 594.351,Z 501.26,A -85,B 0,C 180,E1 -1205.408,E2 -1205.408} C_VEL
LIN {X 0,Y 594.387,Z 501.252,A -85,B 0,C 180,E1 -1207.94,E2 -1207.94} C_VEL
LIN {X 0,Y 594.38,Z 501.261,A -85,B 0,C 180,E1 -1210.822,E2 -1210.822} C_VEL
LIN {X 0,Y 594.381,Z 501.257,A -85,B 0,C 180,E1 -1213.297,E2 -1213.297} C_VEL
LIN {X 0,Y 594.375,Z 501.254,A -85,B 0,C 180,E1 -1216.158,E2 -1216.158} C_VEL
LIN {X 0,Y 594.377,Z 501.26,A -85,B 0,C 180,E1 -1219.176,E2 -1219.176} C_VEL
LIN {X 0,Y 594.381,Z 501.253,A -85,B 0,C 180,E1 -1222.059,E2 -1222.059} C_VEL
LIN {X 0,Y 594.383,Z 501.258,A -85,B 0,C 180,E1 -1224.67,E2 -1224.67} C_VEL
LIN {X 0,Y 594.371,Z 501.261,A -85,B 0,C 180,E1 -1227.087,E2 -1227.087} C_VEL
LIN {X 0,Y 594.392,Z 501.252,A -85,B 0,C 180,E1 -1229.669,E2 -1229.669} C_VEL
LIN {X 0,Y 594.381,Z 501.257,A -85,B 0,C 180,E1 -1232.54,E2 -1232.54} C_VEL
LIN {X 0,Y 594.377,Z 501.262,A -85,B 0,C 180,E1 -1234.807,E2 -1234.807} C_VEL
LIN {X 0,Y 594.358,Z 501.26,A -85,B 0,C 180,E1 -1237.263,E2 -1237.263} C_VEL
LIN {X 0,Y 594.372,Z 501.254,A -85,B 0,C 180,E1 -1239.946,E2 -1239.946} C_VEL
LIN {X 0,Y 594.384,Z 501.262,A -85,B 0,C 180,E1 -1242.807,E2 -1242.807} C_VEL
LIN {X 0,Y 594.378,Z 501.253,A -85,B 0,C 180,E1 -1245.826,E2 -1245.826} C_VEL
LIN {X 0,Y 594.387,Z 501.255,A -85,B 0,C 180,E1 -1248.404,E2 -1248.404} C_VEL
LIN {X 0,Y 594.397,Z 501.256,A -85,B 0,C 180,E1 -1251.158,E2 -1251.158} C_VEL
LIN {X 0,Y 594.38,Z 501.253,A -85,B 0,C 180,E1 -1253.891,E2 -1253.891} C_VEL
LIN {X 0,Y 594.387,Z 501.259,A -85,B 0,C 180,E1 -1256.611,E2 -1256.611} C_VEL
LIN {X 0,Y 594.421,Z 501.251,A -85,B 0,C 180,E1 -1259.323,E2 -1259.323} C_VEL
LIN {X 0,Y 594.388,Z 501.253,A -85,B 0,C 180,E1 -1262.033,E2 -1262.033} C_VEL
LIN {X 0,Y 594.397,Z 501.261,A -85,B 0,C 180,E1 -1264.748,E2 -1264.748} C_VEL
LIN {X 0,Y 594.411,Z 501.253,A -85,B 0,C 180,E1 -1267.473,E2 -1267.473} C_VEL
LIN {X 0,Y 594.418,Z 501.478,A -85,B 0,C 180,E1 -1268.542,E2 -1268.542} C_VEL
LIN {X 0,Y 594.681,Z 502.72,A -85,B 0,C 180,E1 -1268.645,E2 -1268.645} C_VEL
LIN {X 0,Y 594.667,Z 535.528,A -85,B 0,C 180,E1 -1269.074,E2 -1269.074} C_VEL
LIN {X 0,Y 594.623,Z 548.991,A -85,B 0,C 180,E1 -1269.396,E2 -1269.396} C_VEL
LIN {X 0,Y 594.58,Z 559.393,A -85,B 0,C 180,E1 -1269.756,E2 -1269.756} C_VEL
LIN {X 0,Y 593.96,Z 564.83,A -85,B 0,C 180,E1 -1269.971,E2 -1269.971} C_VEL
LIN {X 0,Y 591.076,Z 573.475,A -85,B 0,C 180,E1 -1270.35,E2 -1270.35} C_VEL
LIN {X 0,Y 588.137,Z 581.789,A -85,B 0,C 180,E1 -1270.798,E2 -1270.798} C_VEL
LIN {X 0,Y 587.431,Z 586.603,A -85,B 0,C 180,E1 -1271.119,E2 -1271.119} C_VEL
LIN {X 0,Y 587.347,Z 596.49,A -85,B 0,C 180,E1 -1271.912,E2 -1271.912} C_VEL
LIN {X 0,Y 587.31,Z 605.427,A -85,B 0,C 180,E1 -1272.79,E2 -1272.79} C_VEL
LIN {X 0,Y 587.24,Z 612.822,A -85,B 0,C 180,E1 -1273.672,E2 -1273.672} C_VEL
LIN {X 0,Y 587.232,Z 620.092,A -85,B 0,C 180,E1 -1274.734,E2 -1274.734} C_VEL
LIN {X 0,Y 587.189,Z 625.031,A -85,B 0,C 180,E1 -1275.623,E2 -1275.623} C_VEL
LIN {X 0,Y 587.165,Z 630.068,A -85,B 0,C 180,E1 -1276.759,E2 -1276.759} C_VEL
LIN {X 0,Y 587.133,Z 634.387,A -85,B 0,C 180,E1 -1278.133,E2 -1278.133} C_VEL
LIN {X 0,Y 587.147,Z 636.206,A -85,B 0,C 180,E1 -1278.988,E2 -1278.988} C_VEL
LIN {X 0,Y 587.118,Z 637.753,A -85,B 0,C 180,E1 -1280.313,E2 -1280.313} C_VEL
LIN {X 0,Y 587.136,Z 638,A -85,B 0,C 180,E1 -1281.045,E2 -1281.045} C_VEL
LIN {X 0,Y 587.135,Z 637.75,A -85,B 0,C 180,E1 -1281.782,E2 -1281.782} C_VEL
LIN {X 0,Y 587.119,Z 636.648,A -85,B 0,C 180,E1 -1282.825,E2 -1282.825} C_VEL
LIN {X 0,Y 587.125,Z 634.233,A -85,B 0,C 180,E1 -1284.016,E2 -1284.016} C_VEL
LIN {X 0,Y 587.175,Z 630.75,A -85,B 0,C 180,E1 -1285.145,E2 -1285.145} C_VEL
LIN {X 0,Y 587.2,Z 625.951,A -85,B 0,C 180,E1 -1286.286,E2 -1286.286} C_VEL
LIN {X 0,Y 587.206,Z 620.072,A -85,B 0,C 180,E1 -1287.362,E2 -1287.362} C_VEL
LIN {X 0,Y 587.265,Z 612.901,A -85,B 0,C 180,E1 -1288.405,E2 -1288.405} C_VEL
LIN {X 0,Y 587.305,Z 604.638,A -85,B 0,C 180,E1 -1289.382,E2 -1289.382} C_VEL
LIN {X 0,Y 587.384,Z 595.169,A -85,B 0,C 180,E1 -1290.294,E2 -1290.294} C_VEL
LIN {X 0,Y 587.46,Z 583.926,A -85,B 0,C 180,E1 -1291.159,E2 -1291.159} C_VEL
LIN {X 0,Y 587.552,Z 572.195,A -85,B 0,C 180,E1 -1291.87,E2 -1291.87} C_VEL
LIN {X 0,Y 587.596,Z 560.619,A -85,B 0,C 180,E1 -1292.418,E2 -1292.418} C_VEL
LIN {X 0,Y 587.674,Z 547.874,A -85,B 0,C 180,E1 -1292.867,E2 -1292.867} C_VEL
LIN {X 0,Y 587.758,Z 533.549,A -85,B 0,C 180,E1 -1293.195,E2 -1293.195} C_VEL
LIN {X 0,Y 587.635,Z 503.517,A -85,B 0,C 180,E1 -1293.586,E2 -1293.586} C_VEL
LIN {X 0,Y 587.374,Z 502.295,A -85,B 0,C 180,E1 -1293.703,E2 -1293.703} C_VEL
LIN {X 0,Y 587.353,Z 502.131,A -85,B 0,C 180,E1 -1295.896,E2 -1295.896} C_VEL
LIN {X 0,Y 587.328,Z 502.132,A -85,B 0,C 180,E1 -1298.48,E2 -1298.48} C_VEL
LIN {X 0,Y 587.334,Z 502.138,A -85,B 0,C 180,E1 -1301.158,E2 -1301.158} C_VEL
LIN {X 0,Y 587.331,Z 502.131,A -85,B 0,C 180,E1 -1304.115,E2 -1304.115} C_VEL
LIN {X 0,Y 587.334,Z 502.134,A -85,B 0,C 180,E1 -1306.997,E2 -1306.997} C_VEL
LIN {X 0,Y 587.324,Z 502.133,A -85,B 0,C 180,E1 -1309.982,E2 -1309.982} C_VEL
LIN {X 0,Y 587.345,Z 502.129,A -85,B 0,C 180,E1 -1312.393,E2 -1312.393} C_VEL
LIN {X 0,Y 587.361,Z 502.132,A -85,B 0,C 180,E1 -1315.781,E2 -1315.781} C_VEL
LIN {X 0,Y 587.349,Z 502.129,A -85,B 0,C 180,E1 -1318.232,E2 -1318.232} C_VEL
LIN {X 0,Y 587.351,Z 502.13,A -85,B 0,C 180,E1 -1320.867,E2 -1320.867} C_VEL
LIN {X 0,Y 587.36,Z 502.133,A -85,B 0,C 180,E1 -1323.82,E2 -1323.82} C_VEL
LIN {X 0,Y 587.332,Z 502.134,A -85,B 0,C 180,E1 -1325.994,E2 -1325.994} C_VEL
LIN {X 0,Y 587.324,Z 502.133,A -85,B 0,C 180,E1 -1328.226,E2 -1328.226} C_VEL
LIN {X 0,Y 587.35,Z 502.132,A -85,B 0,C 180,E1 -1331.152,E2 -1331.152} C_VEL
LIN {X 0,Y 587.326,Z 502.135,A -85,B 0,C 180,E1 -1334.025,E2 -1334.025} C_VEL
LIN {X 0,Y 587.364,Z 502.129,A -85,B 0,C 180,E1 -1336.155,E2 -1336.155} C_VEL
LIN {X 0,Y 587.344,Z 502.13,A -85,B 0,C 180,E1 -1338.963,E2 -1338.963} C_VEL
LIN {X 0,Y 587.368,Z 502.136,A -85,B 0,C 180,E1 -1341.745,E2 -1341.745} C_VEL
LIN {X 0,Y 587.355,Z 502.128,A -85,B 0,C 180,E1 -1344.507,E2 -1344.507} C_VEL
LIN {X 0,Y 587.371,Z 502.129,A -85,B 0,C 180,E1 -1347.257,E2 -1347.257} C_VEL
LIN {X 0,Y 587.388,Z 502.13,A -85,B 0,C 180,E1 -1350,E2 -1350} C_VEL
LIN {X 0,Y 587.37,Z 502.126,A -85,B 0,C 180,E1 -1352.743,E2 -1352.743} C_VEL
LIN {X 0,Y 587.357,Z 502.133,A -85,B 0,C 180,E1 -1355.493,E2 -1355.493} C_VEL
LIN {X 0,Y 587.347,Z 502.132,A -85,B 0,C 180,E1 -1358.255,E2 -1358.255} C_VEL
LIN {X 0,Y 587.354,Z 502.129,A -85,B 0,C 180,E1 -1361.133,E2 -1361.133} C_VEL
LIN {X 0,Y 587.37,Z 502.13,A -85,B 0,C 180,E1 -1364.26,E2 -1364.26} C_VEL
LIN {X 0,Y 587.355,Z 502.131,A -85,B 0,C 180,E1 -1367.405,E2 -1367.405} C_VEL
LIN {X 0,Y 587.329,Z 502.135,A -85,B 0,C 180,E1 -1370.304,E2 -1370.304} C_VEL
LIN {X 0,Y 587.318,Z 502.133,A -85,B 0,C 180,E1 -1373.258,E2 -1373.258} C_VEL
LIN {X 0,Y 587.333,Z 502.134,A -85,B 0,C 180,E1 -1375.516,E2 -1375.516} C_VEL
LIN {X 0,Y 587.35,Z 502.136,A -85,B 0,C 180,E1 -1377.817,E2 -1377.817} C_VEL
LIN {X 0,Y 587.341,Z 502.132,A -85,B 0,C 180,E1 -1380.51,E2 -1380.51} C_VEL
LIN {X 0,Y 587.335,Z 502.132,A -85,B 0,C 180,E1 -1383.396,E2 -1383.396} C_VEL
LIN {X 0,Y 587.29,Z 502.144,A -85,B 0,C 180,E1 -1385.899,E2 -1385.899} C_VEL
LIN {X 0,Y 587.333,Z 502.134,A -85,B 0,C 180,E1 -1388.478,E2 -1388.478} C_VEL
LIN {X 0,Y 587.336,Z 502.13,A -85,B 0,C 180,E1 -1391.156,E2 -1391.156} C_VEL
LIN {X 0,Y 587.333,Z 502.141,A -85,B 0,C 180,E1 -1394.113,E2 -1394.113} C_VEL
LIN {X 0,Y 587.31,Z 502.133,A -85,B 0,C 180,E1 -1396.993,E2 -1396.993} C_VEL
LIN {X 0,Y 587.315,Z 502.136,A -85,B 0,C 180,E1 -1399.745,E2 -1399.745} C_VEL
LIN {X 0,Y 587.34,Z 502.136,A -85,B 0,C 180,E1 -1402.392,E2 -1402.392} C_VEL
LIN {X 0,Y 587.347,Z 502.129,A -85,B 0,C 180,E1 -1404.945,E2 -1404.945} C_VEL
LIN {X 0,Y 587.335,Z 502.13,A -85,B 0,C 180,E1 -1407.42,E2 -1407.42} C_VEL
LIN {X 0,Y 587.341,Z 502.133,A -85,B 0,C 180,E1 -1409.83,E2 -1409.83} C_VEL
LIN {X 0,Y 587.345,Z 502.139,A -85,B 0,C 180,E1 -1412.306,E2 -1412.306} C_VEL
LIN {X 0,Y 587.336,Z 502.137,A -85,B 0,C 180,E1 -1414.483,E2 -1414.483} C_VEL
LIN {X 0,Y 587.333,Z 502.131,A -85,B 0,C 180,E1 -1417.486,E2 -1417.486} C_VEL
LIN {X 0,Y 587.325,Z 502.133,A -85,B 0,C 180,E1 -1419.695,E2 -1419.695} C_VEL
LIN {X 0,Y 587.351,Z 502.134,A -85,B 0,C 180,E1 -1422.594,E2 -1422.594} C_VEL
LIN {X 0,Y 587.355,Z 502.129,A -85,B 0,C 180,E1 -1425.739,E2 -1425.739} C_VEL
LIN {X 0,Y 587.334,Z 502.139,A -85,B 0,C 180,E1 -1428.263,E2 -1428.263} C_VEL
LIN {X 0,Y 587.339,Z 502.131,A -85,B 0,C 180,E1 -1431.051,E2 -1431.051} C_VEL
LIN {X 0,Y 587.366,Z 502.126,A -85,B 0,C 180,E1 -1433.264,E2 -1433.264} C_VEL
LIN {X 0,Y 587.31,Z 502.135,A -85,B 0,C 180,E1 -1435.882,E2 -1435.882} C_VEL
LIN {X 0,Y 587.359,Z 502.13,A -85,B 0,C 180,E1 -1437.943,E2 -1437.943} C_VEL
LIN {X 0,Y 587.389,Z 502.131,A -85,B 0,C 180,E1 -1440.685,E2 -1440.685} C_VEL
LIN {X 0,Y 587.329,Z 502.131,A -85,B 0,C 180,E1 -1443.43,E2 -1443.43} C_VEL
LIN {X 0,Y 587.351,Z 502.128,A -85,B 0,C 180,E1 -1445.493,E2 -1445.493} C_VEL
LIN {X 0,Y 587.364,Z 502.132,A -85,B 0,C 180,E1 -1448.255,E2 -1448.255} C_VEL
LIN {X 0,Y 587.337,Z 502.132,A -85,B 0,C 180,E1 -1451.134,E2 -1451.134} C_VEL
LIN {X 0,Y 587.35,Z 502.129,A -85,B 0,C 180,E1 -1453.846,E2 -1453.846} C_VEL
LIN {X 0,Y 587.353,Z 502.135,A -85,B 0,C 180,E1 -1456.819,E2 -1456.819} C_VEL
LIN {X 0,Y 587.336,Z 502.13,A -85,B 0,C 180,E1 -1459.575,E2 -1459.575} C_VEL
LIN {X 0,Y 587.316,Z 502.133,A -85,B 0,C 180,E1 -1461.774,E2 -1461.774} C_VEL
LIN {X 0,Y 587.344,Z 502.139,A -85,B 0,C 180,E1 -1464.759,E2 -1464.759} C_VEL
LIN {X 0,Y 587.322,Z 502.137,A -85,B 0,C 180,E1 -1467.046,E2 -1467.046} C_VEL
LIN {X 0,Y 587.345,Z 502.13,A -85,B 0,C 180,E1 -1469.379,E2 -1469.379} C_VEL
LIN {X 0,Y 587.348,Z 502.128,A -85,B 0,C 180,E1 -1471.838,E2 -1471.838} C_VEL
LIN {X 0,Y 587.352,Z 502.132,A -85,B 0,C 180,E1 -1474.35,E2 -1474.35} C_VEL
LIN {X 0,Y 587.346,Z 502.139,A -85,B 0,C 180,E1 -1476.747,E2 -1476.747} C_VEL
LIN {X 0,Y 587.341,Z 502.132,A -85,B 0,C 180,E1 -1479.36,E2 -1479.36} C_VEL
LIN {X 0,Y 587.328,Z 502.132,A -85,B 0,C 180,E1 -1482.108,E2 -1482.108} C_VEL
LIN {X 0,Y 587.31,Z 502.14,A -85,B 0,C 180,E1 -1485.089,E2 -1485.089} C_VEL
LIN {X 0,Y 587.348,Z 502.128,A -85,B 0,C 180,E1 -1487.928,E2 -1487.928} C_VEL
LIN {X 0,Y 587.332,Z 502.139,A -85,B 0,C 180,E1 -1491.058,E2 -1491.058} C_VEL
LIN {X 0,Y 587.35,Z 502.133,A -85,B 0,C 180,E1 -1493.292,E2 -1493.292} C_VEL
LIN {X 0,Y 587.357,Z 502.128,A -85,B 0,C 180,E1 -1495.781,E2 -1495.781} C_VEL
LIN {X 0,Y 587.35,Z 502.13,A -85,B 0,C 180,E1 -1498.232,E2 -1498.232} C_VEL
LIN {X 0,Y 587.347,Z 502.139,A -85,B 0,C 180,E1 -1500.867,E2 -1500.867} C_VEL
LIN {X 0,Y 587.383,Z 502.319,A -85,B 0,C 180,E1 -1502.257,E2 -1502.257} C_VEL
LIN {X 0,Y 588.187,Z 506.95,A -85,B 0,C 180,E1 -1502.997,E2 -1502.997} C_VEL
LIN {X 0,Y 587.995,Z 525.495,A -85,B 0,C 180,E1 -1505.649,E2 -1505.649} C_VEL
LIN {X 0,Y 587.846,Z 544.018,A -85,B 0,C 180,E1 -1508.247,E2 -1508.247} C_VEL
LIN {X 0,Y 587.681,Z 563.024,A -85,B 0,C 180,E1 -1510.865,E2 -1510.865} C_VEL
LIN {X 0,Y 587.554,Z 583.734,A -85,B 0,C 180,E1 -1513.675,E2 -1513.675} C_VEL
LIN {X 0,Y 587.423,Z 606.24,A -85,B 0,C 180,E1 -1516.685,E2 -1516.685} C_VEL
LIN {X 0,Y 587.329,Z 626.364,A -85,B 0,C 180,E1 -1519.333,E2 -1519.333} C_VEL
LIN {X 0,Y 587.543,Z 628.526,A -85,B 0,C 180,E1 -1519.403,E2 -1519.403} C_VEL
LIN {X 0,Y 587.551,Z 704.154,A -85,B 0,C 180,E1 -1520.338,E2 -1520.338} C_VEL
LIN {X 0,Y 587.5,Z 713.425,A -85,B 0,C 180,E1 -1520.533,E2 -1520.533} C_VEL
LIN {X 0,Y 587.445,Z 721.898,A -85,B 0,C 180,E1 -1520.792,E2 -1520.792} C_VEL
LIN {X 0,Y 587.419,Z 730.399,A -85,B 0,C 180,E1 -1521.139,E2 -1521.139} C_VEL
LIN {X 0,Y 587.395,Z 738.728,A -85,B 0,C 180,E1 -1521.572,E2 -1521.572} C_VEL
LIN {X 0,Y 587.335,Z 746.768,A -85,B 0,C 180,E1 -1522.091,E2 -1522.091} C_VEL
LIN {X 0,Y 587.29,Z 754.419,A -85,B 0,C 180,E1 -1522.695,E2 -1522.695} C_VEL
LIN {X 0,Y 587.281,Z 762.809,A -85,B 0,C 180,E1 -1523.512,E2 -1523.512} C_VEL
LIN {X 0,Y 587.238,Z 769.432,A -85,B 0,C 180,E1 -1524.334,E2 -1524.334} C_VEL
LIN {X 0,Y 587.186,Z 774.986,A -85,B 0,C 180,E1 -1525.194,E2 -1525.194} C_VEL
LIN {X 0,Y 587.209,Z 780.147,A -85,B 0,C 180,E1 -1526.226,E2 -1526.226} C_VEL
LIN {X 0,Y 587.158,Z 782.788,A -85,B 0,C 180,E1 -1526.912,E2 -1526.912} C_VEL
LIN {X 0,Y 587.138,Z 785.68,A -85,B 0,C 180,E1 -1527.942,E2 -1527.942} C_VEL
LIN {X 0,Y 587.146,Z 786.935,A -85,B 0,C 180,E1 -1528.628,E2 -1528.628} C_VEL
LIN {X 0,Y 587.138,Z 787.712,A -85,B 0,C 180,E1 -1529.314,E2 -1529.314} C_VEL
LIN {X 0,Y 587.134,Z 788,A -85,B 0,C 180,E1 -1530,E2 -1530} C_VEL
LIN {X 0,Y 587.138,Z 787.712,A -85,B 0,C 180,E1 -1530.686,E2 -1530.686} C_VEL
LIN {X 0,Y 587.146,Z 786.936,A -85,B 0,C 180,E1 -1531.372,E2 -1531.372} C_VEL
LIN {X 0,Y 587.138,Z 785.68,A -85,B 0,C 180,E1 -1532.058,E2 -1532.058} C_VEL
LIN {X 0,Y 587.158,Z 782.788,A -85,B 0,C 180,E1 -1533.087,E2 -1533.087} C_VEL
LIN {X 0,Y 587.21,Z 780.147,A -85,B 0,C 180,E1 -1533.774,E2 -1533.774} C_VEL
LIN {X 0,Y 587.186,Z 774.987,A -85,B 0,C 180,E1 -1534.806,E2 -1534.806} C_VEL
LIN {X 0,Y 587.238,Z 769.433,A -85,B 0,C 180,E1 -1535.666,E2 -1535.666} C_VEL
LIN {X 0,Y 587.269,Z 761.287,A -85,B 0,C 180,E1 -1536.645,E2 -1536.645} C_VEL
LIN {X 0,Y 587.29,Z 754.42,A -85,B 0,C 180,E1 -1537.305,E2 -1537.305} C_VEL
LIN {X 0,Y 587.335,Z 746.769,A -85,B 0,C 180,E1 -1537.909,E2 -1537.909} C_VEL
LIN {X 0,Y 587.395,Z 738.73,A -85,B 0,C 180,E1 -1538.428,E2 -1538.428} C_VEL
LIN {X 0,Y 587.418,Z 730.401,A -85,B 0,C 180,E1 -1538.861,E2 -1538.861} C_VEL
LIN {X 0,Y 587.445,Z 721.899,A -85,B 0,C 180,E1 -1539.207,E2 -1539.207} C_VEL
LIN {X 0,Y 587.512,Z 711.764,A -85,B 0,C 180,E1 -1539.51,E2 -1539.51} C_VEL
LIN {X 0,Y 587.574,Z 700.081,A -85,B 0,C 180,E1 -1539.726,E2 -1539.726} C_VEL
LIN {X 0,Y 587.44,Z 627.698,A -85,B 0,C 180,E1 -1540.61,E2 -1540.61} C_VEL
LIN {X 0,Y 587.343,Z 626.142,A -85,B 0,C 180,E1 -1540.688,E2 -1540.688} C_VEL
LIN {X 0,Y 587.428,Z 604.917,A -85,B 0,C 180,E1 -1543.491,E2 -1543.491} C_VEL
LIN {X 0,Y 587.555,Z 583.735,A -85,B 0,C 180,E1 -1546.325,E2 -1546.325} C_VEL
LIN {X 0,Y 587.681,Z 563.026,A -85,B 0,C 180,E1 -1549.135,E2 -1549.135} C_VEL
LIN {X 0,Y 587.871,Z 542.695,A -85,B 0,C 180,E1 -1551.937,E2 -1551.937} C_VEL
LIN {X 0,Y 588.043,Z 522.837,A -85,B 0,C 180,E1 -1554.727,E2 -1554.727} C_VEL
LIN {X 0,Y 588.187,Z 506.951,A -85,B 0,C 180,E1 -1557.003,E2 -1557.003} C_VEL
LIN {X 0,Y 587.371,Z 502.254,A -85,B 0,C 180,E1 -1557.768,E2 -1557.768} C_VEL
LIN {X 0,Y 587.34,Z 502.134,A -85,B 0,C 180,E1 -1560.51,E2 -1560.51} C_VEL
LIN {X 0,Y 587.336,Z 502.139,A -85,B 0,C 180,E1 -1563.111,E2 -1563.111} C_VEL
LIN {X 0,Y 587.315,Z 502.133,A -85,B 0,C 180,E1 -1565.897,E2 -1565.897} C_VEL
LIN {X 0,Y 587.332,Z 502.134,A -85,B 0,C 180,E1 -1568.478,E2 -1568.478} C_VEL
LIN {X 0,Y 587.335,Z 502.138,A -85,B 0,C 180,E1 -1571.156,E2 -1571.156} C_VEL
LIN {X 0,Y 587.328,Z 502.132,A -85,B 0,C 180,E1 -1574.114,E2 -1574.114} C_VEL
LIN {X 0,Y 587.316,Z 502.142,A -85,B 0,C 180,E1 -1576.994,E2 -1576.994} C_VEL
LIN {X 0,Y 587.315,Z 502.133,A -85,B 0,C 180,E1 -1579.746,E2 -1579.746} C_VEL
LIN {X 0,Y 587.339,Z 502.132,A -85,B 0,C 180,E1 -1582.392,E2 -1582.392} C_VEL
LIN {X 0,Y 587.347,Z 502.139,A -85,B 0,C 180,E1 -1584.946,E2 -1584.946} C_VEL
LIN {X 0,Y 587.333,Z 502.133,A -85,B 0,C 180,E1 -1587.421,E2 -1587.421} C_VEL
LIN {X 0,Y 587.339,Z 502.13,A -85,B 0,C 180,E1 -1589.83,E2 -1589.83} C_VEL
LIN {X 0,Y 587.342,Z 502.131,A -85,B 0,C 180,E1 -1592.306,E2 -1592.306} C_VEL
LIN {X 0,Y 587.336,Z 502.134,A -85,B 0,C 180,E1 -1594.484,E2 -1594.484} C_VEL
LIN {X 0,Y 587.333,Z 502.133,A -85,B 0,C 180,E1 -1597.486,E2 -1597.486} C_VEL
LIN {X 0,Y 587.327,Z 502.132,A -85,B 0,C 180,E1 -1599.695,E2 -1599.695} C_VEL
LIN {X 0,Y 587.35,Z 502.134,A -85,B 0,C 180,E1 -1602.594,E2 -1602.594} C_VEL
LIN {X 0,Y 587.354,Z 502.128,A -85,B 0,C 180,E1 -1605.739,E2 -1605.739} C_VEL
LIN {X 0,Y 587.351,Z 502.139,A -85,B 0,C 180,E1 -1608.859,E2 -1608.859} C_VEL
LIN {X 0,Y 587.364,Z 502.127,A -85,B 0,C 180,E1 -1611.745,E2 -1611.745} C_VEL
LIN {X 0,Y 587.359,Z 502.133,A -85,B 0,C 180,E1 -1614.507,E2 -1614.507} C_VEL
LIN {X 0,Y 587.378,Z 502.129,A -85,B 0,C 180,E1 -1617.257,E2 -1617.257} C_VEL
LIN {X 0,Y 587.373,Z 502.126,A -85,B 0,C 180,E1 -1620,E2 -1620} C_VEL
LIN {X 0,Y 587.377,Z 502.135,A -85,B 0,C 180,E1 -1622.743,E2 -1622.743} C_VEL
LIN {X 0,Y 587.359,Z 502.13,A -85,B 0,C 180,E1 -1625.493,E2 -1625.493} C_VEL
LIN {X 0,Y 587.377,Z 502.293,A -85,B 0,C 180,E1 -1628.385,E2 -1628.385} C_VEL
LIN {X 0,Y 587.615,Z 503.423,A -85,B 0,C 180,E1 -1628.501,E2 -1628.501} C_VEL
LIN {X 0,Y 587.782,Z 517.396,A -85,B 0,C 180,E1 -1628.683,E2 -1628.683} C_VEL
LIN {X 0,Y 587.732,Z 536.201,A -85,B 0,C 180,E1 -1628.943,E2 -1628.943} C_VEL
LIN {X 0,Y 587.674,Z 550.162,A -85,B 0,C 180,E1 -1629.291,E2 -1629.291} C_VEL
LIN {X 0,Y 587.59,Z 561.95,A -85,B 0,C 180,E1 -1629.727,E2 -1629.727} C_VEL
LIN {X 0,Y 587.534,Z 572.744,A -85,B 0,C 180,E1 -1630.25,E2 -1630.25} C_VEL
LIN {X 0,Y 587.481,Z 582.844,A -85,B 0,C 180,E1 -1630.861,E2 -1630.861} C_VEL
LIN {X 0,Y 587.431,Z 586.603,A -85,B 0,C 180,E1 -1631.119,E2 -1631.119} C_VEL
LIN {X 0,Y 586.729,Z 591.309,A -85,B 0,C 180,E1 -1631.463,E2 -1631.463} C_VEL
LIN {X 0,Y 583.778,Z 598.66,A -85,B 0,C 180,E1 -1632.05,E2 -1632.05} C_VEL
LIN {X 0,Y 580.859,Z 605.466,A -85,B 0,C 180,E1 -1632.7,E2 -1632.7} C_VEL
LIN {X 0,Y 580.21,Z 609.317,A -85,B 0,C 180,E1 -1633.137,E2 -1633.137} C_VEL
LIN {X 0,Y 580.169,Z 617.773,A -85,B 0,C 180,E1 -1634.287,E2 -1634.287} C_VEL
LIN {X 0,Y 580.133,Z 622.662,A -85,B 0,C 180,E1 -1635.098,E2 -1635.098} C_VEL
LIN {X 0,Y 580.11,Z 627.923,A -85,B 0,C 180,E1 -1636.18,E2 -1636.18} C_VEL
LIN {X 0,Y 580.063,Z 632.001,A -85,B 0,C 180,E1 -1637.268,E2 -1637.268} C_VEL
LIN {X 0,Y 580.038,Z 634.986,A -85,B 0,C 180,E1 -1638.363,E2 -1638.363} C_VEL
LIN {X 0,Y 580.048,Z 636.417,A -85,B 0,C 180,E1 -1639.096,E2 -1639.096} C_VEL
LIN {X 0,Y 580.019,Z 637.376,A -85,B 0,C 180,E1 -1639.833,E2 -1639.833} C_VEL
LIN {X 0,Y 580.033,Z 637.994,A -85,B 0,C 180,E1 -1641.1,E2 -1641.1} C_VEL
LIN {X 0,Y 580.025,Z 637.568,A -85,B 0,C 180,E1 -1642.063,E2 -1642.063} C_VEL
LIN {X 0,Y 580.037,Z 636.484,A -85,B 0,C 180,E1 -1642.953,E2 -1642.953} C_VEL
LIN {X 0,Y 580.046,Z 633.52,A -85,B 0,C 180,E1 -1644.328,E2 -1644.328} C_VEL
LIN {X 0,Y 580.081,Z 629.706,A -85,B 0,C 180,E1 -1645.474,E2 -1645.474} C_VEL
LIN {X 0,Y 580.129,Z 624.518,A -85,B 0,C 180,E1 -1646.631,E2 -1646.631} C_VEL
LIN {X 0,Y 580.132,Z 618.876,A -85,B 0,C 180,E1 -1647.627,E2 -1647.627} C_VEL
LIN {X 0,Y 580.197,Z 612.202,A -85,B 0,C 180,E1 -1648.586,E2 -1648.586} C_VEL
LIN {X 0,Y 580.249,Z 604.408,A -85,B 0,C 180,E1 -1649.509,E2 -1649.509} C_VEL
LIN {X 0,Y 580.36,Z 594.45,A -85,B 0,C 180,E1 -1650.471,E2 -1650.471} C_VEL
LIN {X 0,Y 580.437,Z 583.922,A -85,B 0,C 180,E1 -1651.284,E2 -1651.284} C_VEL
LIN {X 0,Y 580.551,Z 572.584,A -85,B 0,C 180,E1 -1651.981,E2 -1651.981} C_VEL
LIN {X 0,Y 580.632,Z 562.183,A -85,B 0,C 180,E1 -1652.488,E2 -1652.488} C_VEL
LIN {X 0,Y 580.729,Z 551.462,A -85,B 0,C 180,E1 -1652.894,E2 -1652.894} C_VEL
LIN {X 0,Y 580.762,Z 540.5,A -85,B 0,C 180,E1 -1653.2,E2 -1653.2} C_VEL
LIN {X 0,Y 580.824,Z 527.498,A -85,B 0,C 180,E1 -1653.433,E2 -1653.433} C_VEL
LIN {X 0,Y 580.752,Z 504.96,A -85,B 0,C 180,E1 -1653.715,E2 -1653.715} C_VEL
LIN {X 0,Y 580.404,Z 503.482,A -85,B 0,C 180,E1 -1653.794,E2 -1653.794} C_VEL
LIN {X 0,Y 580.322,Z 503.016,A -85,B 0,C 180,E1 -1653.959,E2 -1653.959} C_VEL
LIN {X 0,Y 580.292,Z 503.01,A -85,B 0,C 180,E1 -1656.402,E2 -1656.402} C_VEL
LIN {X 0,Y 580.304,Z 503.016,A -85,B 0,C 180,E1 -1659.188,E2 -1659.188} C_VEL
LIN {X 0,Y 580.31,Z 503.009,A -85,B 0,C 180,E1 -1661.767,E2 -1661.767} C_VEL
LIN {X 0,Y 580.265,Z 503.011,A -85,B 0,C 180,E1 -1664.627,E2 -1664.627} C_VEL
LIN {X 0,Y 580.288,Z 503.017,A -85,B 0,C 180,E1 -1667.296,E2 -1667.296} C_VEL
LIN {X 0,Y 580.296,Z 503.008,A -85,B 0,C 180,E1 -1670.069,E2 -1670.069} C_VEL
LIN {X 0,Y 580.298,Z 503.011,A -85,B 0,C 180,E1 -1673.067,E2 -1673.067} C_VEL
LIN {X 0,Y 580.316,Z 503.006,A -85,B 0,C 180,E1 -1676.146,E2 -1676.146} C_VEL
LIN {X 0,Y 580.283,Z 503.009,A -85,B 0,C 180,E1 -1678.616,E2 -1678.616} C_VEL
LIN {X 0,Y 580.295,Z 503.01,A -85,B 0,C 180,E1 -1681.025,E2 -1681.025} C_VEL
LIN {X 0,Y 580.293,Z 503.015,A -85,B 0,C 180,E1 -1683.667,E2 -1683.667} C_VEL
LIN {X 0,Y 580.301,Z 503.014,A -85,B 0,C 180,E1 -1685.684,E2 -1685.684} C_VEL
LIN {X 0,Y 580.288,Z 503.008,A -85,B 0,C 180,E1 -1688.695,E2 -1688.695} C_VEL
LIN {X 0,Y 580.3,Z 503.008,A -85,B 0,C 180,E1 -1690.914,E2 -1690.914} C_VEL
LIN {X 0,Y 580.276,Z 503.016,A -85,B 0,C 180,E1 -1693.826,E2 -1693.826} C_VEL
LIN {X 0,Y 580.33,Z 503.007,A -85,B 0,C 180,E1 -1695.984,E2 -1695.984} C_VEL
LIN {X 0,Y 580.31,Z 503.005,A -85,B 0,C 180,E1 -1698.827,E2 -1698.827} C_VEL
LIN {X 0,Y 580.331,Z 503.013,A -85,B 0,C 180,E1 -1701.644,E2 -1701.644} C_VEL
LIN {X 0,Y 580.32,Z 503.005,A -85,B 0,C 180,E1 -1704.44,E2 -1704.44} C_VEL
LIN {X 0,Y 580.338,Z 503.005,A -85,B 0,C 180,E1 -1707.224,E2 -1707.224} C_VEL
LIN {X 0,Y 580.358,Z 503.005,A -85,B 0,C 180,E1 -1710,E2 -1710} C_VEL
LIN {X 0,Y 580.337,Z 503.002,A -85,B 0,C 180,E1 -1712.777,E2 -1712.777} C_VEL
LIN {X 0,Y 580.323,Z 503.01,A -85,B 0,C 180,E1 -1715.56,E2 -1715.56} C_VEL
LIN {X 0,Y 580.316,Z 503.007,A -85,B 0,C 180,E1 -1718.356,E2 -1718.356} C_VEL
LIN {X 0,Y 580.306,Z 503.007,A -85,B 0,C 180,E1 -1721.191,E2 -1721.191} C_VEL
LIN {X 0,Y 580.331,Z 503.01,A -85,B 0,C 180,E1 -1724.017,E2 -1724.017} C_VEL
LIN {X 0,Y 580.317,Z 503.004,A -85,B 0,C 180,E1 -1726.913,E2 -1726.913} C_VEL
LIN {X 0,Y 580.307,Z 503.015,A -85,B 0,C 180,E1 -1729.822,E2 -1729.822} C_VEL
LIN {X 0,Y 580.293,Z 503.007,A -85,B 0,C 180,E1 -1732.802,E2 -1732.802} C_VEL
LIN {X 0,Y 580.308,Z 503.006,A -85,B 0,C 180,E1 -1735.079,E2 -1735.079} C_VEL
LIN {X 0,Y 580.302,Z 503.013,A -85,B 0,C 180,E1 -1738.185,E2 -1738.185} C_VEL
LIN {X 0,Y 580.289,Z 503.009,A -85,B 0,C 180,E1 -1740.694,E2 -1740.694} C_VEL
LIN {X 0,Y 580.304,Z 503.007,A -85,B 0,C 180,E1 -1743.316,E2 -1743.316} C_VEL
LIN {X 0,Y 580.245,Z 503.019,A -85,B 0,C 180,E1 -1745.755,E2 -1745.755} C_VEL
LIN {X 0,Y 580.289,Z 503.017,A -85,B 0,C 180,E1 -1748.145,E2 -1748.145} C_VEL
LIN {X 0,Y 580.299,Z 503.007,A -85,B 0,C 180,E1 -1750.842,E2 -1750.842} C_VEL
LIN {X 0,Y 580.287,Z 503.011,A -85,B 0,C 180,E1 -1753.656,E2 -1753.656} C_VEL
LIN {X 0,Y 580.273,Z 503.013,A -85,B 0,C 180,E1 -1756.608,E2 -1756.608} C_VEL
LIN {X 0,Y 580.296,Z 503.007,A -85,B 0,C 180,E1 -1759.156,E2 -1759.156} C_VEL
LIN {X 0,Y 580.287,Z 503.014,A -85,B 0,C 180,E1 -1761.926,E2 -1761.926} C_VEL
LIN {X 0,Y 580.304,Z 503.012,A -85,B 0,C 180,E1 -1764.456,E2 -1764.456} C_VEL
LIN {X 0,Y 580.286,Z 503.009,A -85,B 0,C 180,E1 -1766.974,E2 -1766.974} C_VEL
LIN {X 0,Y 580.303,Z 503.006,A -85,B 0,C 180,E1 -1769.425,E2 -1769.425} C_VEL
LIN {X 0,Y 580.314,Z 503.013,A -85,B 0,C 180,E1 -1772.136,E2 -1772.136} C_VEL
LIN {X 0,Y 580.303,Z 503.007,A -85,B 0,C 180,E1 -1774.92,E2 -1774.92} C_VEL
LIN {X 0,Y 580.267,Z 503.015,A -85,B 0,C 180,E1 -1777.947,E2 -1777.947} C_VEL
LIN {X 0,Y 580.31,Z 503.007,A -85,B 0,C 180,E1 -1780.913,E2 -1780.913} C_VEL
LIN {X 0,Y 580.274,Z 503.012,A -85,B 0,C 180,E1 -1783.825,E2 -1783.825} C_VEL
LIN {X 0,Y 580.317,Z 503.009,A -85,B 0,C 180,E1 -1785.983,E2 -1785.983} C_VEL
LIN {X 0,Y 580.294,Z 503.011,A -85,B 0,C 180,E1 -1788.826,E2 -1788.826} C_VEL
LIN {X 0,Y 580.327,Z 503.004,A -85,B 0,C 180,E1 -1791.644,E2 -1791.644} C_VEL
LIN {X 0,Y 580.317,Z 503.015,A -85,B 0,C 180,E1 -1794.44,E2 -1794.44} C_VEL
LIN {X 0,Y 580.339,Z 503.002,A -85,B 0,C 180,E1 -1797.223,E2 -1797.223} C_VEL
LIN {X 0,Y 580.343,Z 503.004,A -85,B 0,C 180,E1 -1800,E2 -1800} C_VEL
LIN {X 0,Y 580.339,Z 503.008,A -85,B 0,C 180,E1 -1802.776,E2 -1802.776} C_VEL
LIN {X 0,Y 580.317,Z 503.004,A -85,B 0,C 180,E1 -1805.56,E2 -1805.56} C_VEL
LIN {X 0,Y 580.327,Z 503.01,A -85,B 0,C 180,E1 -1808.356,E2 -1808.356} C_VEL
LIN {X 0,Y 580.289,Z 503.009,A -85,B 0,C 180,E1 -1811.191,E2 -1811.191} C_VEL
LIN {X 0,Y 580.316,Z 503.006,A -85,B 0,C 180,E1 -1814.017,E2 -1814.017} C_VEL
LIN {X 0,Y 580.303,Z 503.012,A -85,B 0,C 180,E1 -1816.915,E2 -1816.915} C_VEL
LIN {X 0,Y 580.299,Z 503.007,A -85,B 0,C 180,E1 -1819.822,E2 -1819.822} C_VEL
LIN {X 0,Y 580.266,Z 503.012,A -85,B 0,C 180,E1 -1822.053,E2 -1822.053} C_VEL
LIN {X 0,Y 580.301,Z 503.01,A -85,B 0,C 180,E1 -1825.08,E2 -1825.08} C_VEL
LIN {X 0,Y 580.312,Z 503.005,A -85,B 0,C 180,E1 -1827.864,E2 -1827.864} C_VEL
LIN {X 0,Y 580.291,Z 503.018,A -85,B 0,C 180,E1 -1830.698,E2 -1830.698} C_VEL
LIN {X 0,Y 580.297,Z 503.009,A -85,B 0,C 180,E1 -1833.317,E2 -1833.317} C_VEL
LIN {X 0,Y 580.321,Z 503.004,A -85,B 0,C 180,E1 -1835.768,E2 -1835.768} C_VEL
LIN {X 0,Y 580.282,Z 503.01,A -85,B 0,C 180,E1 -1838.147,E2 -1838.147} C_VEL
LIN {X 0,Y 580.294,Z 503.018,A -85,B 0,C 180,E1 -1840.844,E2 -1840.844} C_VEL
LIN {X 0,Y 580.272,Z 503.01,A -85,B 0,C 180,E1 -1843.658,E2 -1843.658} C_VEL
LIN {X 0,Y 580.281,Z 503.015,A -85,B 0,C 180,E1 -1846.609,E2 -1846.609} C_VEL
LIN {X 0,Y 580.296,Z 503.013,A -85,B 0,C 180,E1 -1849.157,E2 -1849.157} C_VEL
LIN {X 0,Y 580.288,Z 503.008,A -85,B 0,C 180,E1 -1851.927,E2 -1851.927} C_VEL
LIN {X 0,Y 580.282,Z 503.012,A -85,B 0,C 180,E1 -1854.456,E2 -1854.456} C_VEL
LIN {X 0,Y 580.289,Z 503.019,A -85,B 0,C 180,E1 -1856.976,E2 -1856.976} C_VEL
LIN {X 0,Y 580.3,Z 503.012,A -85,B 0,C 180,E1 -1859.426,E2 -1859.426} C_VEL
LIN {X 0,Y 580.351,Z 503.205,A -85,B 0,C 180,E1 -1862.085,E2 -1862.085} C_VEL
LIN {X 0,Y 581.317,Z 508.166,A -85,B 0,C 180,E1 -1862.846,E2 -1862.846} C_VEL
LIN {X 0,Y 581.143,Z 525.928,A -85,B 0,C 180,E1 -1865.405,E2 -1865.405} C_VEL
LIN {X 0,Y 580.973,Z 544.018,A -85,B 0,C 180,E1 -1867.976,E2 -1867.976} C_VEL
LIN {X 0,Y 580.739,Z 563.723,A -85,B 0,C 180,E1 -1870.724,E2 -1870.724} C_VEL
LIN {X 0,Y 580.555,Z 585.058,A -85,B 0,C 180,E1 -1873.653,E2 -1873.653} C_VEL
LIN {X 0,Y 580.415,Z 606.24,A -85,B 0,C 180,E1 -1876.521,E2 -1876.521} C_VEL
LIN {X 0,Y 580.312,Z 626.431,A -85,B 0,C 180,E1 -1879.208,E2 -1879.208} C_VEL
LIN {X 0,Y 580.592,Z 629.348,A -85,B 0,C 180,E1 -1879.284,E2 -1879.284} C_VEL
LIN {X 0,Y 580.562,Z 704.154,A -85,B 0,C 180,E1 -1880.221,E2 -1880.221} C_VEL
LIN {X 0,Y 580.487,Z 713.426,A -85,B 0,C 180,E1 -1880.417,E2 -1880.417} C_VEL
LIN {X 0,Y 580.46,Z 721.9,A -85,B 0,C 180,E1 -1880.681,E2 -1880.681} C_VEL
LIN {X 0,Y 580.42,Z 730.402,A -85,B 0,C 180,E1 -1881.031,E2 -1881.031} C_VEL
LIN {X 0,Y 580.362,Z 738.73,A -85,B 0,C 180,E1 -1881.469,E2 -1881.469} C_VEL
LIN {X 0,Y 580.31,Z 746.77,A -85,B 0,C 180,E1 -1881.994,E2 -1881.994} C_VEL
LIN {X 0,Y 580.239,Z 754.42,A -85,B 0,C 180,E1 -1882.606,E2 -1882.606} C_VEL
LIN {X 0,Y 580.22,Z 763,A -85,B 0,C 180,E1 -1883.454,E2 -1883.454} C_VEL
LIN {X 0,Y 580.173,Z 769.433,A -85,B 0,C 180,E1 -1884.265,E2 -1884.265} C_VEL
LIN {X 0,Y 580.097,Z 774.987,A -85,B 0,C 180,E1 -1885.135,E2 -1885.135} C_VEL
LIN {X 0,Y 580.136,Z 780.148,A -85,B 0,C 180,E1 -1886.18,E2 -1886.18} C_VEL
LIN {X 0,Y 580.072,Z 782.788,A -85,B 0,C 180,E1 -1886.875,E2 -1886.875} C_VEL
LIN {X 0,Y 580.038,Z 785.68,A -85,B 0,C 180,E1 -1887.917,E2 -1887.917} C_VEL
LIN {X 0,Y 580.045,Z 786.936,A -85,B 0,C 180,E1 -1888.611,E2 -1888.611} C_VEL
LIN {X 0,Y 580.038,Z 787.711,A -85,B 0,C 180,E1 -1889.306,E2 -1889.306} C_VEL
LIN {X 0,Y 580.034,Z 788,A -85,B 0,C 180,E1 -1890,E2 -1890} C_VEL
LIN {X 0,Y 580.038,Z 787.712,A -85,B 0,C 180,E1 -1890.694,E2 -1890.694} C_VEL
LIN {X 0,Y 580.045,Z 786.936,A -85,B 0,C 180,E1 -1891.388,E2 -1891.388} C_VEL
LIN {X 0,Y 580.038,Z 785.681,A -85,B 0,C 180,E1 -1892.083,E2 -1892.083} C_VEL
LIN {X 0,Y 580.072,Z 782.789,A -85,B 0,C 180,E1 -1893.125,E2 -1893.125} C_VEL
LIN {X 0,Y 580.122,Z 780.148,A -85,B 0,C 180,E1 -1893.82,E2 -1893.82} C_VEL
LIN {X 0,Y 580.097,Z 774.988,A -85,B 0,C 180,E1 -1894.865,E2 -1894.865} C_VEL
LIN {X 0,Y 580.173,Z 769.434,A -85,B 0,C 180,E1 -1895.735,E2 -1895.735} C_VEL
LIN {X 0,Y 580.209,Z 761.949,A -85,B 0,C 180,E1 -1896.659,E2 -1896.659} C_VEL
LIN {X 0,Y 580.239,Z 754.421,A -85,B 0,C 180,E1 -1897.394,E2 -1897.394} C_VEL
LIN {X 0,Y 580.31,Z 746.771,A -85,B 0,C 180,E1 -1898.006,E2 -1898.006} C_VEL
LIN {X 0,Y 580.362,Z 738.732,A -85,B 0,C 180,E1 -1898.531,E2 -1898.531} C_VEL
LIN {X 0,Y 580.42,Z 730.404,A -85,B 0,C 180,E1 -1898.969,E2 -1898.969} C_VEL
LIN {X 0,Y 580.438,Z 721.9,A -85,B 0,C 180,E1 -1899.32,E2 -1899.32} C_VEL
LIN {X 0,Y 580.511,Z 711.764,A -85,B 0,C 180,E1 -1899.626,E2 -1899.626} C_VEL
LIN {X 0,Y 580.602,Z 700.081,A -85,B 0,C 180,E1 -1899.844,E2 -1899.844} C_VEL
LIN {X 0,Y 580.512,Z 628.529,A -85,B 0,C 180,E1 -1900.727,E2 -1900.727} C_VEL
LIN {X 0,Y 580.312,Z 626.416,A -85,B 0,C 180,E1 -1900.792,E2 -1900.792} C_VEL
LIN {X 0,Y 580.415,Z 606.241,A -85,B 0,C 180,E1 -1903.479,E2 -1903.479} C_VEL
LIN {X 0,Y 580.58,Z 583.735,A -85,B 0,C 180,E1 -1906.527,E2 -1906.527} C_VEL
LIN {X 0,Y 580.804,Z 562.251,A -85,B 0,C 180,E1 -1909.478,E2 -1909.478} C_VEL
LIN {X 0,Y 581.01,Z 540.047,A -85,B 0,C 180,E1 -1912.584,E2 -1912.584} C_VEL
LIN {X 0,Y 581.257,Z 518.866,A -85,B 0,C 180,E1 -1915.61,E2 -1915.61} C_VEL
LIN {X 0,Y 581.317,Z 508.142,A -85,B 0,C 180,E1 -1917.154,E2 -1917.154} C_VEL
LIN {X 0,Y 580.319,Z 503.083,A -85,B 0,C 180,E1 -1917.905,E2 -1917.905} C_VEL
LIN {X 0,Y 580.29,Z 503.015,A -85,B 0,C 180,E1 -1920.696,E2 -1920.696} C_VEL
LIN {X 0,Y 580.3,Z 503.012,A -85,B 0,C 180,E1 -1923.316,E2 -1923.316} C_VEL
LIN {X 0,Y 580.272,Z 503.011,A -85,B 0,C 180,E1 -1925.76,E2 -1925.76} C_VEL
LIN {X 0,Y 580.287,Z 503.009,A -85,B 0,C 180,E1 -1928.145,E2 -1928.145} C_VEL
LIN {X 0,Y 580.298,Z 503.016,A -85,B 0,C 180,E1 -1930.842,E2 -1930.842} C_VEL
LIN {X 0,Y 580.285,Z 503.01,A -85,B 0,C 180,E1 -1933.656,E2 -1933.656} C_VEL
LIN {X 0,Y 580.279,Z 503.014,A -85,B 0,C 180,E1 -1936.608,E2 -1936.608} C_VEL
LIN {X 0,Y 580.295,Z 503.014,A -85,B 0,C 180,E1 -1939.156,E2 -1939.156} C_VEL
LIN {X 0,Y 580.284,Z 503.009,A -85,B 0,C 180,E1 -1941.926,E2 -1941.926} C_VEL
LIN {X 0,Y 580.303,Z 503.009,A -85,B 0,C 180,E1 -1944.456,E2 -1944.456} C_VEL
LIN {X 0,Y 580.284,Z 503.018,A -85,B 0,C 180,E1 -1946.975,E2 -1946.975} C_VEL
LIN {X 0,Y 580.302,Z 503.009,A -85,B 0,C 180,E1 -1949.426,E2 -1949.426} C_VEL
LIN {X 0,Y 580.311,Z 503.006,A -85,B 0,C 180,E1 -1952.136,E2 -1952.136} C_VEL
LIN {X 0,Y 580.302,Z 503.017,A -85,B 0,C 180,E1 -1954.92,E2 -1954.92} C_VEL
LIN {X 0,Y 580.266,Z 503.011,A -85,B 0,C 180,E1 -1957.947,E2 -1957.947} C_VEL
LIN {X 0,Y 580.308,Z 503.016,A -85,B 0,C 180,E1 -1960.914,E2 -1960.914} C_VEL
LIN {X 0,Y 580.276,Z 503.01,A -85,B 0,C 180,E1 -1963.826,E2 -1963.826} C_VEL
LIN {X 0,Y 580.273,Z 503.018,A -85,B 0,C 180,E1 -1966.696,E2 -1966.696} C_VEL
LIN {X 0,Y 580.298,Z 503.009,A -85,B 0,C 180,E1 -1969.533,E2 -1969.533} C_VEL
LIN {X 0,Y 580.332,Z 503.006,A -85,B 0,C 180,E1 -1972.345,E2 -1972.345} C_VEL
LIN {X 0,Y 580.338,Z 503.008,A -85,B 0,C 180,E1 -1975.137,E2 -1975.137} C_VEL
LIN {X 0,Y 580.33,Z 503.004,A -85,B 0,C 180,E1 -1977.918,E2 -1977.918} C_VEL
LIN {X 0,Y 580.362,Z 503.008,A -85,B 0,C 180,E1 -1980.694,E2 -1980.694} C_VEL
LIN {X 0,Y 580.285,Z 503.011,A -85,B 0,C 180,E1 -1983.472,E2 -1983.472} C_VEL
LIN {X 0,Y 580.325,Z 503.007,A -85,B 0,C 180,E1 -1985.56,E2 -1985.56} C_VEL
LIN {X 0,Y 580.339,Z 503.127,A -85,B 0,C 180,E1 -1988.225,E2 -1988.225} C_VEL
LIN {X 0,Y 580.549,Z 504.193,A -85,B 0,C 180,E1 -1988.353,E2 -1988.353} C_VEL
LIN {X 0,Y 580.861,Z 507.844,A -85,B 0,C 180,E1 -1988.414,E2 -1988.414} C_VEL
LIN {X 0,Y 580.795,Z 535.756,A -85,B 0,C 180,E1 -1988.788,E2 -1988.788} C_VEL
LIN {X 0,Y 580.731,Z 549.149,A -85,B 0,C 180,E1 -1989.118,E2 -1989.118} C_VEL
LIN {X 0,Y 580.654,Z 561.731,A -85,B 0,C 180,E1 -1989.58,E2 -1989.58} C_VEL
LIN {X 0,Y 580.555,Z 572.583,A -85,B 0,C 180,E1 -1990.11,E2 -1990.11} C_VEL
LIN {X 0,Y 580.463,Z 582.721,A -85,B 0,C 180,E1 -1990.729,E2 -1990.729} C_VEL
LIN {X 0,Y 580.368,Z 592.876,A -85,B 0,C 180,E1 -1991.491,E2 -1991.491} C_VEL
LIN {X 0,Y 580.273,Z 602.876,A -85,B 0,C 180,E1 -1992.415,E2 -1992.415} C_VEL
LIN {X 0,Y 580.21,Z 609.317,A -85,B 0,C 180,E1 -1993.137,E2 -1993.137} C_VEL
LIN {X 0,Y 579.561,Z 612.964,A -85,B 0,C 180,E1 -1993.593,E2 -1993.593} C_VEL
LIN {X 0,Y 576.644,Z 618.507,A -85,B 0,C 180,E1 -1994.356,E2 -1994.356} C_VEL
LIN {X 0,Y 573.7,Z 623.403,A -85,B 0,C 180,E1 -1995.168,E2 -1995.168} C_VEL
LIN {X 0,Y 573.02,Z 626.025,A -85,B 0,C 180,E1 -1995.694,E2 -1995.694} C_VEL
LIN {X 0,Y 572.999,Z 631.056,A -85,B 0,C 180,E1 -1996.929,E2 -1996.929} C_VEL
LIN {X 0,Y 572.96,Z 633.881,A -85,B 0,C 180,E1 -1997.858,E2 -1997.858} C_VEL
LIN {X 0,Y 572.956,Z 636.588,A -85,B 0,C 180,E1 -1999.183,E2 -1999.183} C_VEL
LIN {X 0,Y 572.944,Z 637.617,A -85,B 0,C 180,E1 -2000.088,E2 -2000.088} C_VEL
LIN {X 0,Y 572.955,Z 637.968,A -85,B 0,C 180,E1 -2001.218,E2 -2001.218} C_VEL
LIN {X 0,Y 572.929,Z 637.293,A -85,B 0,C 180,E1 -2002.351,E2 -2002.351} C_VEL
LIN {X 0,Y 572.928,Z 636.271,A -85,B 0,C 180,E1 -2003.113,E2 -2003.113} C_VEL
LIN {X 0,Y 572.964,Z 633.802,A -85,B 0,C 180,E1 -2004.263,E2 -2004.263} C_VEL
LIN {X 0,Y 573.002,Z 630.127,A -85,B 0,C 180,E1 -2005.422,E2 -2005.422} C_VEL
LIN {X 0,Y 573.037,Z 625.766,A -85,B 0,C 180,E1 -2006.455,E2 -2006.455} C_VEL
LIN {X 0,Y 573.064,Z 619.677,A -85,B 0,C 180,E1 -2007.579,E2 -2007.579} C_VEL
LIN {X 0,Y 573.123,Z 613.006,A -85,B 0,C 180,E1 -2008.571,E2 -2008.571} C_VEL
LIN {X 0,Y 573.206,Z 605.562,A -85,B 0,C 180,E1 -2009.483,E2 -2009.483} C_VEL
LIN {X 0,Y 573.314,Z 596.746,A -85,B 0,C 180,E1 -2010.376,E2 -2010.376} C_VEL
LIN {X 0,Y 573.406,Z 586.977,A -85,B 0,C 180,E1 -2011.188,E2 -2011.188} C_VEL
LIN {X 0,Y 573.557,Z 575.422,A -85,B 0,C 180,E1 -2011.957,E2 -2011.957} C_VEL
LIN {X 0,Y 573.668,Z 563.578,A -85,B 0,C 180,E1 -2012.567,E2 -2012.567} C_VEL
LIN {X 0,Y 573.751,Z 553.261,A -85,B 0,C 180,E1 -2012.979,E2 -2012.979} C_VEL
LIN {X 0,Y 573.802,Z 541.846,A -85,B 0,C 180,E1 -2013.316,E2 -2013.316} C_VEL
LIN {X 0,Y 573.889,Z 530.192,A -85,B 0,C 180,E1 -2013.546,E2 -2013.546} C_VEL
LIN {X 0,Y 573.854,Z 506.277,A -85,B 0,C 180,E1 -2013.852,E2 -2013.852} C_VEL
LIN {X 0,Y 573.379,Z 504.444,A -85,B 0,C 180,E1 -2013.932,E2 -2013.932} C_VEL
LIN {X 0,Y 573.285,Z 503.936,A -85,B 0,C 180,E1 -2014.039,E2 -2014.039} C_VEL
LIN {X 0,Y 573.249,Z 503.895,A -85,B 0,C 180,E1 -2017.167,E2 -2017.167} C_VEL
LIN {X 0,Y 573.244,Z 503.892,A -85,B 0,C 180,E1 -2019.608,E2 -2019.608} C_VEL
LIN {X 0,Y 573.239,Z 503.887,A -85,B 0,C 180,E1 -2022.643,E2 -2022.643} C_VEL
LIN {X 0,Y 573.237,Z 503.892,A -85,B 0,C 180,E1 -2025.668,E2 -2025.668} C_VEL
LIN {X 0,Y 573.244,Z 503.886,A -85,B 0,C 180,E1 -2028.545,E2 -2028.545} C_VEL
LIN {X 0,Y 573.248,Z 503.894,A -85,B 0,C 180,E1 -2031.3,E2 -2031.3} C_VEL
LIN {X 0,Y 573.212,Z 503.891,A -85,B 0,C 180,E1 -2034.019,E2 -2034.019} C_VEL
LIN {X 0,Y 573.269,Z 503.882,A -85,B 0,C 180,E1 -2036.519,E2 -2036.519} C_VEL
LIN {X 0,Y 573.235,Z 503.891,A -85,B 0,C 180,E1 -2039.118,E2 -2039.118} C_VEL
LIN {X 0,Y 573.266,Z 503.886,A -85,B 0,C 180,E1 -2041.969,E2 -2041.969} C_VEL
LIN {X 0,Y 573.255,Z 503.884,A -85,B 0,C 180,E1 -2044.591,E2 -2044.591} C_VEL
LIN {X 0,Y 573.238,Z 503.895,A -85,B 0,C 180,E1 -2047.663,E2 -2047.663} C_VEL
LIN {X 0,Y 573.27,Z 503.882,A -85,B 0,C 180,E1 -2050.671,E2 -2050.671} C_VEL
LIN {X 0,Y 573.249,Z 503.895,A -85,B 0,C 180,E1 -2053.622,E2 -2053.622} C_VEL
LIN {X 0,Y 573.278,Z 503.889,A -85,B 0,C 180,E1 -2055.808,E2 -2055.808} C_VEL
LIN {X 0,Y 573.268,Z 503.882,A -85,B 0,C 180,E1 -2058.745,E2 -2058.745} C_VEL
LIN {X 0,Y 573.287,Z 503.888,A -85,B 0,C 180,E1 -2061.541,E2 -2061.541} C_VEL
LIN {X 0,Y 573.287,Z 503.881,A -85,B 0,C 180,E1 -2064.372,E2 -2064.372} C_VEL
LIN {X 0,Y 573.315,Z 503.884,A -85,B 0,C 180,E1 -2067.893,E2 -2067.893} C_VEL
LIN {X 0,Y 573.332,Z 503.874,A -85,B 0,C 180,E1 -2070.702,E2 -2070.702} C_VEL
LIN {X 0,Y 573.305,Z 503.878,A -85,B 0,C 180,E1 -2072.811,E2 -2072.811} C_VEL
LIN {X 0,Y 573.29,Z 503.887,A -85,B 0,C 180,E1 -2075.628,E2 -2075.628} C_VEL
LIN {X 0,Y 573.26,Z 503.885,A -85,B 0,C 180,E1 -2078.46,E2 -2078.46} C_VEL
LIN {X 0,Y 573.278,Z 503.884,A -85,B 0,C 180,E1 -2081.312,E2 -2081.312} C_VEL
LIN {X 0,Y 573.287,Z 503.882,A -85,B 0,C 180,E1 -2084.424,E2 -2084.424} C_VEL
LIN {X 0,Y 573.264,Z 503.883,A -85,B 0,C 180,E1 -2087.111,E2 -2087.111} C_VEL
LIN {X 0,Y 573.254,Z 503.892,A -85,B 0,C 180,E1 -2090.076,E2 -2090.076} C_VEL
LIN {X 0,Y 573.238,Z 503.886,A -85,B 0,C 180,E1 -2093.099,E2 -2093.099} C_VEL
LIN {X 0,Y 573.255,Z 503.886,A -85,B 0,C 180,E1 -2095.409,E2 -2095.409} C_VEL
LIN {X 0,Y 573.255,Z 503.894,A -85,B 0,C 180,E1 -2098.028,E2 -2098.028} C_VEL
LIN {X 0,Y 573.234,Z 503.887,A -85,B 0,C 180,E1 -2100.882,E2 -2100.882} C_VEL
LIN {X 0,Y 573.263,Z 503.886,A -85,B 0,C 180,E1 -2103.523,E2 -2103.523} C_VEL
LIN {X 0,Y 573.214,Z 503.9,A -85,B 0,C 180,E1 -2106.051,E2 -2106.051} C_VEL
LIN {X 0,Y 573.248,Z 503.886,A -85,B 0,C 180,E1 -2108.7,E2 -2108.7} C_VEL
LIN {X 0,Y 573.252,Z 503.887,A -85,B 0,C 180,E1 -2111.595,E2 -2111.595} C_VEL
LIN {X 0,Y 573.237,Z 503.893,A -85,B 0,C 180,E1 -2114.332,E2 -2114.332} C_VEL
LIN {X 0,Y 573.237,Z 503.887,A -85,B 0,C 180,E1 -2117.358,E2 -2117.358} C_VEL
LIN {X 0,Y 573.244,Z 503.892,A -85,B 0,C 180,E1 -2120.392,E2 -2120.392} C_VEL
LIN {X 0,Y 573.251,Z 503.885,A -85,B 0,C 180,E1 -2123.077,E2 -2123.077} C_VEL
LIN {X 0,Y 573.27,Z 503.885,A -85,B 0,C 180,E1 -2125.671,E2 -2125.671} C_VEL
LIN {X 0,Y 573.245,Z 503.896,A -85,B 0,C 180,E1 -2128.184,E2 -2128.184} C_VEL
LIN {X 0,Y 573.264,Z 503.887,A -85,B 0,C 180,E1 -2130.634,E2 -2130.634} C_VEL
LIN {X 0,Y 573.264,Z 503.883,A -85,B 0,C 180,E1 -2133.5,E2 -2133.5} C_VEL
LIN {X 0,Y 573.226,Z 503.896,A -85,B 0,C 180,E1 -2136.134,E2 -2136.134} C_VEL
LIN {X 0,Y 573.254,Z 503.884,A -85,B 0,C 180,E1 -2139.173,E2 -2139.173} C_VEL
LIN {X 0,Y 573.231,Z 503.887,A -85,B 0,C 180,E1 -2141.411,E2 -2141.411} C_VEL
LIN {X 0,Y 573.25,Z 503.885,A -85,B 0,C 180,E1 -2143.621,E2 -2143.621} C_VEL
LIN {X 0,Y 573.229,Z 503.895,A -85,B 0,C 180,E1 -2146.529,E2 -2146.529} C_VEL
LIN {X 0,Y 573.253,Z 503.889,A -85,B 0,C 180,E1 -2148.744,E2 -2148.744} C_VEL
LIN {X 0,Y 573.299,Z 503.879,A -85,B 0,C 180,E1 -2151.54,E2 -2151.54} C_VEL
LIN {X 0,Y 573.284,Z 503.89,A -85,B 0,C 180,E1 -2154.371,E2 -2154.371} C_VEL
LIN {X 0,Y 573.301,Z 503.88,A -85,B 0,C 180,E1 -2157.892,E2 -2157.892} C_VEL
LIN {X 0,Y 573.328,Z 503.882,A -85,B 0,C 180,E1 -2160.702,E2 -2160.702} C_VEL
LIN {X 0,Y 573.232,Z 503.887,A -85,B 0,C 180,E1 -2163.514,E2 -2163.514} C_VEL
LIN {X 0,Y 573.284,Z 503.881,A -85,B 0,C 180,E1 -2165.628,E2 -2165.628} C_VEL
LIN {X 0,Y 573.298,Z 503.888,A -85,B 0,C 180,E1 -2168.459,E2 -2168.459} C_VEL
LIN {X 0,Y 573.261,Z 503.884,A -85,B 0,C 180,E1 -2171.312,E2 -2171.312} C_VEL
LIN {X 0,Y 573.263,Z 503.887,A -85,B 0,C 180,E1 -2174.193,E2 -2174.193} C_VEL
LIN {X 0,Y 573.25,Z 503.888,A -85,B 0,C 180,E1 -2177.112,E2 -2177.112} C_VEL
LIN {X 0,Y 573.248,Z 503.887,A -85,B 0,C 180,E1 -2180.077,E2 -2180.077} C_VEL
LIN {X 0,Y 573.229,Z 503.892,A -85,B 0,C 180,E1 -2182.338,E2 -2182.338} C_VEL
LIN {X 0,Y 573.25,Z 503.886,A -85,B 0,C 180,E1 -2185.41,E2 -2185.41} C_VEL
LIN {X 0,Y 573.256,Z 503.885,A -85,B 0,C 180,E1 -2188.032,E2 -2188.032} C_VEL
LIN {X 0,Y 573.236,Z 503.895,A -85,B 0,C 180,E1 -2190.885,E2 -2190.885} C_VEL
LIN {X 0,Y 573.281,Z 503.881,A -85,B 0,C 180,E1 -2193.529,E2 -2193.529} C_VEL
LIN {X 0,Y 573.254,Z 503.885,A -85,B 0,C 180,E1 -2196.048,E2 -2196.048} C_VEL
LIN {X 0,Y 573.243,Z 503.894,A -85,B 0,C 180,E1 -2198.701,E2 -2198.701} C_VEL
LIN {X 0,Y 573.247,Z 503.886,A -85,B 0,C 180,E1 -2201.596,E2 -2201.596} C_VEL
LIN {X 0,Y 573.229,Z 503.89,A -85,B 0,C 180,E1 -2204.334,E2 -2204.334} C_VEL
LIN {X 0,Y 573.239,Z 503.889,A -85,B 0,C 180,E1 -2207.359,E2 -2207.359} C_VEL
LIN {X 0,Y 573.244,Z 503.888,A -85,B 0,C 180,E1 -2210.394,E2 -2210.394} C_VEL
LIN {X 0,Y 573.253,Z 503.893,A -85,B 0,C 180,E1 -2213.079,E2 -2213.079} C_VEL
LIN {X 0,Y 573.264,Z 503.885,A -85,B 0,C 180,E1 -2215.672,E2 -2215.672} C_VEL
LIN {X 0,Y 573.246,Z 503.887,A -85,B 0,C 180,E1 -2218.186,E2 -2218.186} C_VEL
LIN {X 0,Y 573.262,Z 503.891,A -85,B 0,C 180,E1 -2220.635,E2 -2220.635} C_VEL
LIN {X 0,Y 573.279,Z 504.061,A -85,B 0,C 180,E1 -2221.91,E2 -2221.91} C_VEL
LIN {X 0,Y 574.412,Z 510.425,A -85,B 0,C 180,E1 -2222.887,E2 -2222.887} C_VEL
LIN {X 0,Y 574.271,Z 526.363,A -85,B 0,C 180,E1 -2225.154,E2 -2225.154} C_VEL
LIN {X 0,Y 574.097,Z 542.695,A -85,B 0,C 180,E1 -2227.508,E2 -2227.508} C_VEL
LIN {X 0,Y 573.806,Z 564.41,A -85,B 0,C 180,E1 -2230.578,E2 -2230.578} C_VEL
LIN {X 0,Y 573.595,Z 585.07,A -85,B 0,C 180,E1 -2233.451,E2 -2233.451} C_VEL
LIN {X 0,Y 573.402,Z 606.24,A -85,B 0,C 180,E1 -2236.353,E2 -2236.353} C_VEL
LIN {X 0,Y 573.251,Z 626.428,A -85,B 0,C 180,E1 -2239.073,E2 -2239.073} C_VEL
LIN {X 0,Y 573.469,Z 628.56,A -85,B 0,C 180,E1 -2239.14,E2 -2239.14} C_VEL
LIN {X 0,Y 573.592,Z 676.82,A -85,B 0,C 180,E1 -2239.744,E2 -2239.744} C_VEL
LIN {X 0,Y 573.555,Z 705.452,A -85,B 0,C 180,E1 -2240.122,E2 -2240.122} C_VEL
LIN {X 0,Y 573.534,Z 715.917,A -85,B 0,C 180,E1 -2240.367,E2 -2240.367} C_VEL
LIN {X 0,Y 573.454,Z 726.621,A -85,B 0,C 180,E1 -2240.744,E2 -2240.744} C_VEL
LIN {X 0,Y 573.343,Z 737.235,A -85,B 0,C 180,E1 -2241.275,E2 -2241.275} C_VEL
LIN {X 0,Y 573.284,Z 745.55,A -85,B 0,C 180,E1 -2241.807,E2 -2241.807} C_VEL
LIN {X 0,Y 573.214,Z 753.408,A -85,B 0,C 180,E1 -2242.426,E2 -2242.426} C_VEL
LIN {X 0,Y 573.164,Z 760.802,A -85,B 0,C 180,E1 -2243.14,E2 -2243.14} C_VEL
LIN {X 0,Y 573.137,Z 768.191,A -85,B 0,C 180,E1 -2244.017,E2 -2244.017} C_VEL
LIN {X 0,Y 573.005,Z 774.987,A -85,B 0,C 180,E1 -2245.075,E2 -2245.075} C_VEL
LIN {X 0,Y 573.036,Z 780.148,A -85,B 0,C 180,E1 -2246.132,E2 -2246.132} C_VEL
LIN {X 0,Y 572.992,Z 782.789,A -85,B 0,C 180,E1 -2246.836,E2 -2246.836} C_VEL
LIN {X 0,Y 572.938,Z 785.681,A -85,B 0,C 180,E1 -2247.891,E2 -2247.891} C_VEL
LIN {X 0,Y 572.945,Z 786.936,A -85,B 0,C 180,E1 -2248.594,E2 -2248.594} C_VEL
LIN {X 0,Y 572.938,Z 787.711,A -85,B 0,C 180,E1 -2249.297,E2 -2249.297} C_VEL
LIN {X 0,Y 572.935,Z 788,A -85,B 0,C 180,E1 -2250,E2 -2250} C_VEL
LIN {X 0,Y 572.938,Z 787.711,A -85,B 0,C 180,E1 -2250.703,E2 -2250.703} C_VEL
LIN {X 0,Y 572.945,Z 786.937,A -85,B 0,C 180,E1 -2251.406,E2 -2251.406} C_VEL
LIN {X 0,Y 572.938,Z 785.682,A -85,B 0,C 180,E1 -2252.109,E2 -2252.109} C_VEL
LIN {X 0,Y 572.992,Z 782.79,A -85,B 0,C 180,E1 -2253.164,E2 -2253.164} C_VEL
LIN {X 0,Y 573.024,Z 780.148,A -85,B 0,C 180,E1 -2253.868,E2 -2253.868} C_VEL
LIN {X 0,Y 573.005,Z 774.989,A -85,B 0,C 180,E1 -2254.925,E2 -2254.925} C_VEL
LIN {X 0,Y 573.137,Z 768.191,A -85,B 0,C 180,E1 -2255.983,E2 -2255.983} C_VEL
LIN {X 0,Y 573.16,Z 760.841,A -85,B 0,C 180,E1 -2256.856,E2 -2256.856} C_VEL
LIN {X 0,Y 573.214,Z 753.409,A -85,B 0,C 180,E1 -2257.574,E2 -2257.574} C_VEL
LIN {X 0,Y 573.283,Z 745.55,A -85,B 0,C 180,E1 -2258.193,E2 -2258.193} C_VEL
LIN {X 0,Y 573.4,Z 735.737,A -85,B 0,C 180,E1 -2258.813,E2 -2258.813} C_VEL
LIN {X 0,Y 573.455,Z 724.308,A -85,B 0,C 180,E1 -2259.345,E2 -2259.345} C_VEL
LIN {X 0,Y 573.498,Z 714.256,A -85,B 0,C 180,E1 -2259.678,E2 -2259.678} C_VEL
LIN {X 0,Y 573.555,Z 705.46,A -85,B 0,C 180,E1 -2259.878,E2 -2259.878} C_VEL
LIN {X 0,Y 573.642,Z 644.187,A -85,B 0,C 180,E1 -2260.662,E2 -2260.662} C_VEL
LIN {X 0,Y 573.427,Z 628.204,A -85,B 0,C 180,E1 -2260.865,E2 -2260.865} C_VEL
